	garr_betriebsmeldungen[st_config.i16_meld_startindex + 0] := bm_fuellstand_oeler;
	garr_betriebsmeldungen[st_config.i16_meld_startindex + 1] := FALSE;
	garr_betriebsmeldungen[st_config.i16_meld_startindex + 2] := FALSE;
	garr_betriebsmeldungen[st_config.i16_meld_startindex + 3] := FALSE;
	garr_betriebsmeldungen[st_config.i16_meld_startindex + 4] := FALSE;
	garr_betriebsmeldungen[st_config.i16_meld_startindex + 5] := FALSE;
	garr_betriebsmeldungen[st_config.i16_meld_startindex + 6] := FALSE;
	garr_betriebsmeldungen[st_config.i16_meld_startindex + 7] := FALSE;
	garr_betriebsmeldungen[st_config.i16_meld_startindex + 8] := FALSE;
	garr_betriebsmeldungen[st_config.i16_meld_startindex + 9] := FALSE;
	garr_betriebsmeldungen[st_config.i16_meld_startindex + 10] := FALSE;
	garr_betriebsmeldungen[st_config.i16_meld_startindex + 11] := FALSE;
	garr_betriebsmeldungen[st_config.i16_meld_startindex + 12] := FALSE;
	garr_betriebsmeldungen[st_config.i16_meld_startindex + 13] := FALSE;
	garr_betriebsmeldungen[st_config.i16_meld_startindex + 14] := FALSE;
	garr_betriebsmeldungen[st_config.i16_meld_startindex + 15] := FALSE;
	garr_betriebsmeldungen[st_config.i16_meld_startindex + 16] := FALSE;
	garr_betriebsmeldungen[st_config.i16_meld_startindex + 17] := FALSE;
	garr_betriebsmeldungen[st_config.i16_meld_startindex + 18] := FALSE;
	garr_betriebsmeldungen[st_config.i16_meld_startindex + 19] := FALSE;
END_IF
END_PROGRAM

(* POU Gemeinsamkeiten17xx/Programmbausteine/ST_Schreibe_Persistente_Daten, ST *)
PROGRAM ST_Schreibe_Persistente_Daten
VAR_INPUT
	bExecute			: BOOL;
	bQuit				: BOOL;
	t_schreibintervall		: TIME;
	b_steuerung_ein		: BOOL;
END_VAR
VAR_OUTPUT
	bBusy				: BOOL;
	bError				: BOOL;
	nErrId				: UDINT;
END_VAR
VAR
	fb_write_persistent_data		: FB_WritePersistentData;
	fb_ton_quitt					: TON;
	fb_state_entry				: ST_StateEntry;
	fb_ton_schreiben			: TON;
	fb_get_local_ams_netid		: ST_GetLocalAMSNetID;
	fb_r_trig_execute			: R_TRIG;
	fb_f_trig_steuerung			: F_TRIG;
	sm_fehler_daten_schreiben	: BOOL := FALSE;
	sm_fehler_netid				: BOOL := FALSE;

	gst_manuelles_bestueckprogramm_copy	: struct_bestueckprogramm;
	gst_PersDaten_Copy					: struct_PD;
END_VAR
(* Die Persistenten Daten der Maschine werden in einem wiederkehrenden Zeitintervall in eine Datei im TwinCAT Boot-Ordner geschrieben *)
fb_ton_quitt(IN:= , PT:= t#30s, Q=> , ET=> );
fb_ton_schreiben(IN:= , PT:= t_schreibintervall, Q=> , ET=> );

fb_r_trig_execute(CLK:= bExecute, Q=> );
fb_f_trig_steuerung(CLK:= b_steuerung_ein, Q=> );


fb_state_entry(	i16_pos:= 1 );

CASE fb_state_entry.i16_step OF
(*=======================================================*)
	INIT_OBJ:
		fb_state_entry.i16_next_step := INIT;

(*=======================================================*)
	INIT:
		IF fb_state_entry.E THEN
			bBusy := FALSE;
			bError := FALSE;
			fb_write_persistent_data.START := FALSE;
			fb_ton_schreiben.IN := FALSE;
			fb_get_local_ams_netid.bExecute := FALSE;
			fb_get_local_ams_netid .bQuit := FALSE;
			sm_fehler_daten_schreiben := FALSE;
			sm_fehler_netid := FALSE;
		END_IF

		fb_state_entry.i16_next_step := 20;

(*=======================================================*)
	20:	(* Die AMS-NetID des lokalen PC ermitteln *)
		IF fb_state_entry.E THEN
			fb_get_local_ams_netid.bExecute := TRUE;
		END_IF

		IF fb_get_local_ams_netid.bBusy THEN
			fb_get_local_ams_netid.bExecute := FALSE;
			fb_state_entry.i16_next_step := 30;
		END_IF

(*=======================================================*)
	30:
		IF NOT fb_get_local_ams_netid.bBusy  THEN
			IF NOT fb_get_local_ams_netid.bError THEN
				fb_state_entry.i16_next_step := BEREIT;
			ELSE	(* Fehler *)
				sm_fehler_netid := TRUE;
				fb_state_entry.i16_next_step := FEHLER;
			END_IF
		END_IF

(*=======================================================*)
	BEREIT:	(* Warte auf Freigabeflanke für zyklisches Schreiben der Daten /  Daten sichern, wenn Maschine ausgeschaltet wird *)
		IF 	fb_r_trig_execute.Q OR fb_f_trig_steuerung.Q THEN
			fb_state_entry.i16_next_step := 110;
		END_IF

		(*Schreibe bei einer Änderung*)
		IF	gi16_maschinenstatusinfo <> STATUS_MASCHINE_ARBEITET AND (
			(MEMCMP(ADR(gst_manuelles_bestueckprogramm_copy), ADR(gst_manuelles_bestueckprogramm), SIZEOF(gst_manuelles_bestueckprogramm_copy)) <> 0 ) OR
			(MEMCMP(ADR(gst_PersDaten_Copy), ADR(gst_PersDaten), SIZEOF(gst_PersDaten_Copy)) <> 0 ) 	) THEN
			gst_PersDaten_Copy:=gst_PersDaten;
			gst_manuelles_bestueckprogramm_copy:=gst_manuelles_bestueckprogramm;
			fb_state_entry.i16_next_step := 110;
		END_IF

(*=======================================================*)
	110:	(* Schreibe Persistente Daten *)
		IF fb_state_entry.E THEN
			bBusy := TRUE;
			fb_write_persistent_data.START := TRUE;
		END_IF

		IF fb_write_persistent_data.BUSY THEN
			fb_write_persistent_data.START := FALSE;
			fb_state_entry.i16_next_step := 120;
		END_IF

(*=======================================================*)
	120:	(* Daten wurden geschrieben *)
		IF NOT fb_write_persistent_data.BUSY  THEN
			IF NOT fb_write_persistent_data.ERR THEN
				bBusy := FALSE;
				fb_state_entry.i16_next_step := 100;
			ELSE
				sm_fehler_daten_schreiben := TRUE;
				fb_state_entry.i16_next_step := FEHLER;
			END_IF
		END_IF

(*=======================================================*)
	FEHLER:
		IF fb_state_entry.E THEN
			fb_ton_quitt.IN := TRUE;
			fb_get_local_ams_netid.bExecute := FALSE;
			fb_get_local_ams_netid.bQuit := FALSE;
			bError := TRUE;
		END_IF

		IF  fb_ton_quitt.Q THEN
			fb_ton_quitt.IN := FALSE;
			fb_get_local_ams_netid .bQuit := TRUE;
			fb_state_entry.i16_next_step := INIT;
		END_IF

END_CASE

fb_state_entry(i16_pos:= 2 );

fb_get_local_ams_netid(
	bExecute:= ,
	bQuit:= , 
	bBusy=> , 
	bReady=> , 
	bError=> , 
	nErrId=> , 
	s_ams_netid=> );

fb_write_persistent_data(
	NETID:= '',
	PORT:= 801,
	START:= , 
	TMOUT:= DEFAULT_ADS_TIMEOUT,
	MODE:= SPDM_2PASS,
	BUSY=> , 
	ERR=> , 
	ERRID=> );
END_PROGRAM

(* POU Gemeinsamkeiten17xx/TagReader/ST_Lesen_Schreiben_Tag, ST *)
PROGRAM ST_Lesen_Schreiben_Tag
VAR_INPUT
	st_config					: struct_config;
	st_ctrl_in					: struct_ctrl_in;
END_VAR
VAR_OUTPUT
	st_ctrl_out				: struct_ctrl_out;
END_VAR
VAR
	fb_r_trig_lesen			: R_TRIG;
	fb_r_trig_schreiben		: R_TRIG;
	fb_r_trig_WT_ruecksetzen	: R_TRIG;
	fb_r_trig_auto_lesen		: R_TRIG;
	fb_ton_lesen				: TON;
	fb_ton_auto_lesen				: TON;
	fb_ton_Timeout				: TON;

	fb_state_entry				: ST_StateEntry;
	fb_ton_quitt				: TON;
	fb_r_trig_quittieren			: R_TRIG;
	fb_ton_uez				: TON;

	sm_WT_Nummer_ungueltig				: BOOL := FALSE;
	sm_wt_hat_kein_tag					: BOOL := FALSE;
	bm_kein_WT_im_Aktionsfeld			: BOOL := FALSE;
	bm_Wert_nicht_erlaubt					: BOOL := FALSE;

	i									: INT;

	i16_betriebsart: BOOL;
END_VAR
fb_ton_quitt(IN:= , PT:= t#500ms, Q=> , ET=> );
fb_ton_uez(IN:= , PT:= , Q=>  , ET=> );

fb_ton_lesen(IN:= , PT:= t#500ms, Q=> , ET=> );
fb_r_trig_lesen(CLK:=visu.st_tagreader.b_start_lesen , Q=>);
fb_ton_auto_lesen(IN:=balluff_tag_reader.fb.e_tag_im_aktionsfeld   AND gi16_betriebsart = HAND , PT:= t#500ms, Q=> , ET=> );
fb_r_trig_auto_lesen(CLK:= fb_ton_auto_lesen.Q , Q=>);


fb_r_trig_schreiben(CLK:=visu.st_tagreader.b_start_schreiben , Q=>);
fb_r_trig_WT_ruecksetzen(CLK:=visu.st_tagreader.b_WT_ruecksetzen , Q=>);

visu.st_tagreader.b_tag_im_Aktionsfeld:=balluff_tag_reader.fb.e_tag_im_aktionsfeld;

fb_state_entry(
	i16_next_step:= ,
	i16_pos:= 1,
	s_debugtext:= ,
	E=> ,
	X=> ,
	i16_step=> ,
	i16_last_step=> );

(*wenn Tagreader nicht bereit ist stoppen*)
IF	Balluff_Tag_Reader.fb.fb_state_entry.i16_step<BEREIT OR
	Balluff_Tag_Reader.fb.fb_state_entry.i16_step>=STOP THEN
	fb_state_entry.i16_next_step := STOP;
END_IF

fb_ton_Timeout(IN:= fb_state_entry.i16_step>BEREIT AND fb_state_entry.i16_step<FEHLER, PT:= t#35s, Q=> , ET=> );
IF	fb_ton_Timeout.Q THEN
	fb_state_entry.i16_next_step := FEHLER;
END_IF

CASE fb_state_entry.i16_step OF
(*=======================================================*)
	INIT_OBJ:

		fb_state_entry.i16_next_step := INIT;

(*=======================================================*)
	INIT:
		IF 	fb_state_entry.E THEN
			balluff_tag_reader.st_ctrl.in.b_start_lesen := FALSE;
			balluff_tag_reader.st_ctrl.in.b_start_schreiben := FALSE;

			sm_WT_Nummer_ungueltig:=FALSE;
			sm_wt_hat_kein_tag:=FALSE;

			visu.st_tagreader.b_WT_ruecksetzen:=FALSE;
			visu.st_tagreader.b_start_schreiben:=FALSE;
			visu.st_tagreader.b_start_lesen:=FALSE;
		END_IF

		(*-----------------------Weiterschaltbedingungen----------------------------*)
		fb_state_entry.i16_next_step := BEREIT;

(*=======================================================*)
	BEREIT:	(* Warte auf Start von Kontroller *)

		(*-----------------------Weiterschaltbedingungen----------------------------*)
		IF	balluff_tag_reader.fb.e_tag_im_aktionsfeld   AND gi16_betriebsart = HAND THEN
			IF	fb_r_trig_lesen.Q  OR fb_r_trig_auto_lesen.Q THEN
				fb_state_entry.i16_next_step := 120;
			END_IF

			IF	fb_r_trig_schreiben.Q THEN
				fb_state_entry.i16_next_step := 150;
			END_IF

			IF	fb_r_trig_WT_ruecksetzen.Q THEN
				fb_state_entry.i16_next_step := 200;
			END_IF
		ELSE
			IF	fb_r_trig_WT_ruecksetzen.Q OR
				fb_r_trig_schreiben.Q OR
				fb_r_trig_lesen.Q THEN
				fb_state_entry.i16_next_step := 110;
			END_IF
		END_IF

(*=======================================================*)
	110:
		IF 	fb_state_entry.E THEN
			fb_ton_uez.PT:=t#2000ms ;
			fb_ton_uez.IN:=TRUE ;
			bm_kein_WT_im_Aktionsfeld:=TRUE;
		END_IF

		(*-----------------------Weiterschaltbedingungen----------------------------*)
		IF	fb_ton_uez.Q THEN
			fb_state_entry.i16_next_step := INIT;
			fb_ton_uez.IN:=FALSE ;
			bm_kein_WT_im_Aktionsfeld:=FALSE;
		END_IF

(*=======================================================*)
	120:
		IF 	fb_state_entry.E THEN
			gst_tag_data.Articelnumber:='LESEN';
			gst_tag_data.LastUsedTool:=0;
			IF gst_datensatz.st_md.i16_tag_data_structur_version = 0 THEN
				gst_tag_data.StateParts[0]:=100;
				gst_tag_data.StateParts[1]:=100;
			ELSIF gst_datensatz.st_md.i16_tag_data_structur_version = 1 THEN
				FOR i:= 0 TO 7 BY 1 DO
					gst_tag_data.StateParts[i] := 100;
				END_FOR
			END_IF
			gst_tag_data.WpcNumber:=0;
			fb_ton_lesen.IN:=TRUE;
		END_IF

	(*-----------------------Weiterschaltbedingungen----------------------------*)
	IF	fb_ton_lesen.Q THEN
		fb_ton_lesen.IN:=FALSE;
		fb_state_entry.i16_next_step := 130;
	END_IF

(*=======================================================*)
	130: (* WT-Tag mit RFID-Lesegerät auslesen *)
		IF 	fb_state_entry.E THEN
			balluff_tag_reader.st_ctrl.in.b_start_lesen := TRUE;
			balluff_tag_reader.fb.i16_addresse := 0;
			balluff_tag_reader.fb.i16_anzahl_byte := SIZEOF(gst_tag_data);
		END_IF

		(*-----------------------Weiterschaltbedingungen----------------------------*)
		IF 	balluff_tag_reader.st_ctrl.out.b_fertig AND NOT fb_state_entry.E THEN
			IF gst_datensatz.st_md.i16_tag_data_structur_version = 0 THEN
				gst_tag_data.WpcNumber := balluff_tag_reader.fb.s_lese_daten[0];
				gst_tag_data.StateParts[0] := balluff_tag_reader.fb.s_lese_daten[1];
				gst_tag_data.StateParts[1] := balluff_tag_reader.fb.s_lese_daten[2];

				MEMCPY( ADR(gst_tag_data.Articelnumber), ADR(balluff_tag_reader.fb.s_lese_daten[3]), 50);
				gst_tag_data.LastUsedTool := balluff_tag_reader.fb.s_lese_daten[54];
				MEMCPY( ADR(gst_tag_data.UmlNo_VPE), ADR(balluff_tag_reader.fb.s_lese_daten[55]), 4);

				(*gst_datensatz.st_md.s_aktuelle_artikelnummer := gst_tag_data.Articelnumber;*)
			ELSIF gst_datensatz.st_md.i16_tag_data_structur_version = 1 THEN
				gst_tag_data.WpcNumber := balluff_tag_reader.fb.s_lese_daten[0];
				FOR i:= 0 TO 7 BY 1 DO
					gst_tag_data.StateParts[i] := balluff_tag_reader.fb.s_lese_daten[i + 1];
				END_FOR
				gst_tag_data.AmountPartsOnWpc := balluff_tag_reader.fb.s_lese_daten[10];
				gst_tag_data.LastUsedTool := balluff_tag_reader.fb.s_lese_daten[15];
				MEMCPY( ADR(gst_tag_data.Articelnumber), ADR(balluff_tag_reader.fb.s_lese_daten[20]), 50);
				MEMCPY( ADR(gst_tag_data.UmlNo_VPE), ADR(balluff_tag_reader.fb.s_lese_daten[71]), 4);
			END_IF

			IF 	gst_tag_data.WpcNumber >= 0 AND gst_tag_data.WpcNumber <=50 THEN
				balluff_tag_reader.st_ctrl.in.b_start_lesen := FALSE;
				fb_state_entry.i16_next_step := INIT;
			ELSE
				(* Fehler: Tagnummer ist nicht im gültigem Bereich *)
				balluff_tag_reader.st_ctrl.in.b_start_lesen := FALSE;
				sm_WT_Nummer_ungueltig := TRUE;
				fb_state_entry.i16_next_step := FEHLER;
			END_IF
		END_IF

(*=======================================================*)
	150:	(*Artikelnummer schreiben*)
		IF 	fb_state_entry.E THEN
			IF gst_datensatz.st_md.i16_tag_data_structur_version = 0 THEN
				balluff_tag_reader.st_ctrl.in.b_start_schreiben := TRUE;
	
				balluff_tag_reader.fb.i16_addresse := 3;
				balluff_tag_reader.fb.i16_anzahl_byte := SIZEOF(gst_tag_data.Articelnumber);
				MEMCPY(ADR(balluff_tag_reader.fb.s_schreib_daten),ADR(gst_tag_data.Articelnumber),  50);
			ELSIF gst_datensatz.st_md.i16_tag_data_structur_version = 1 THEN
				balluff_tag_reader.st_ctrl.in.b_start_schreiben := TRUE;
	
				balluff_tag_reader.fb.i16_addresse := 20;
				balluff_tag_reader.fb.i16_anzahl_byte := SIZEOF(gst_tag_data.Articelnumber);
				MEMCPY(ADR(balluff_tag_reader.fb.s_schreib_daten),ADR(gst_tag_data.Articelnumber),  50);
			END_IF
		END_IF

		(*-----------------------Weiterschaltbedingungen----------------------------*)
		IF 	balluff_tag_reader.st_ctrl.out.b_fertig AND NOT fb_state_entry.E THEN
			(* Ok: Daten sind auf dem Tag *)
			balluff_tag_reader.st_ctrl.in.b_start_schreiben := FALSE;
			fb_state_entry.i16_next_step := 155;
		END_IF

(*=======================================================*)
	155:	(*UML_Stueckzaehler schreiben*)
		IF 	fb_state_entry.E THEN
			IF gst_datensatz.st_md.i16_tag_data_structur_version = 0 THEN
				balluff_tag_reader.st_ctrl.in.b_start_schreiben := TRUE;

				balluff_tag_reader.fb.i16_addresse := 55;
				balluff_tag_reader.fb.i16_anzahl_byte := SIZEOF(gst_tag_data.UmlNo_VPE);
				MEMCPY( ADR(balluff_tag_reader.fb.s_schreib_daten), ADR(gst_tag_data.UmlNo_VPE), 4);

			ELSIF gst_datensatz.st_md.i16_tag_data_structur_version = 1 THEN
				balluff_tag_reader.st_ctrl.in.b_start_schreiben := TRUE;

				balluff_tag_reader.fb.i16_addresse := 71;
				balluff_tag_reader.fb.i16_anzahl_byte := SIZEOF(gst_tag_data.UmlNo_VPE);
				MEMCPY(ADR(balluff_tag_reader.fb.s_schreib_daten),ADR(gst_tag_data.UmlNo_VPE),  4);
			END_IF
		END_IF

		(*-----------------------Weiterschaltbedingungen----------------------------*)
		IF 	balluff_tag_reader.st_ctrl.out.b_fertig AND NOT fb_state_entry.E THEN
			(* Ok: Daten sind auf dem Tag *)
			balluff_tag_reader.st_ctrl.in.b_start_schreiben := FALSE;
			fb_state_entry.i16_next_step := 160;
		END_IF

(*=======================================================*)
	160:	(*States schreiben*)
		IF 	fb_state_entry.E THEN
			IF gst_datensatz.st_md.i16_tag_data_structur_version = 0 THEN
				balluff_tag_reader.st_ctrl.in.b_start_schreiben := TRUE;
	
				balluff_tag_reader.fb.i16_addresse := 1;
				balluff_tag_reader.fb.i16_anzahl_byte := 2;
				balluff_tag_reader.fb.s_schreib_daten[0] := DINT_TO_BYTE(gst_tag_data.StateParts[0]);
				balluff_tag_reader.fb.s_schreib_daten[1] := DINT_TO_BYTE(gst_tag_data.StateParts[1]);
			ELSIF gst_datensatz.st_md.i16_tag_data_structur_version = 1 THEN
				balluff_tag_reader.st_ctrl.in.b_start_schreiben := TRUE;
	
				balluff_tag_reader.fb.i16_addresse := 1;
				balluff_tag_reader.fb.i16_anzahl_byte := 8;
				FOR i:= 0 TO 7 BY 1 DO
					balluff_tag_reader.fb.s_schreib_daten[i] := DINT_TO_BYTE(gst_tag_data.StateParts[i]);
				END_FOR
			END_IF
		END_IF

		(*-----------------------Weiterschaltbedingungen----------------------------*)
		IF balluff_tag_reader.st_ctrl.out.b_fertig AND NOT fb_state_entry.E THEN
			(* Ok: Daten sind auf dem Tag *)
			balluff_tag_reader.st_ctrl.in.b_start_schreiben := FALSE;
			fb_state_entry.i16_next_step := 170;
		END_IF

(*=======================================================*)
	170:	(* WT Nummer schreiben *)
		IF	 fb_state_entry.E THEN
			(* Starte Schreib Prozess *)
			balluff_tag_reader.fb.i16_addresse := 0;
			balluff_tag_reader.fb.i16_anzahl_byte := 1;
			balluff_tag_reader.fb.s_schreib_daten[0] := gst_tag_data.WpcNumber;
			balluff_tag_reader.st_ctrl.in.b_start_schreiben := TRUE;
		END_IF

		(*-----------------------Weiterschaltbedingungen----------------------------*)
		IF 	balluff_tag_reader.st_ctrl.out.b_fertig AND NOT fb_state_entry.E THEN
			balluff_tag_reader.st_ctrl.in.b_start_schreiben := FALSE;
			fb_state_entry.i16_next_step := 180;
		END_IF

(*=======================================================*)
	180:	(* letztes benutzes Werkzeug schreiben*)
		IF 	fb_state_entry.E THEN
			(* Starte Schreib Prozess *)
			IF gst_datensatz.st_md.i16_tag_data_structur_version = 0 THEN
				balluff_tag_reader.fb.i16_addresse := 54;
				balluff_tag_reader.fb.i16_anzahl_byte := 1;
				balluff_tag_reader.fb.s_schreib_daten[0] := gst_tag_data.LastUsedTool;
				balluff_tag_reader.st_ctrl.in.b_start_schreiben := TRUE;
			ELSIF gst_datensatz.st_md.i16_tag_data_structur_version = 1 THEN
				balluff_tag_reader.fb.i16_addresse := 15;
				balluff_tag_reader.fb.i16_anzahl_byte := 1;
				balluff_tag_reader.fb.s_schreib_daten[0] := gst_tag_data.LastUsedTool;
				balluff_tag_reader.st_ctrl.in.b_start_schreiben := TRUE;
			END_IF
		END_IF

		(*-----------------------Weiterschaltbedingungen----------------------------*)
		IF 	balluff_tag_reader.st_ctrl.out.b_fertig AND NOT fb_state_entry.E THEN
			balluff_tag_reader.st_ctrl.in.b_start_schreiben := FALSE;
			IF gst_datensatz.st_md.i16_tag_data_structur_version = 0 THEN
				fb_state_entry.i16_next_step := 120;
			ELSIF gst_datensatz.st_md.i16_tag_data_structur_version = 1 THEN
				fb_state_entry.i16_next_step := 190;
			END_IF
		END_IF

(*=======================================================*)
	190:	(* Anzahl ISK auf WT *)
		IF 	fb_state_entry.E THEN
			(* Starte Schreib Prozess *)
			balluff_tag_reader.fb.i16_addresse := 10;
			balluff_tag_reader.fb.i16_anzahl_byte := 1;
			balluff_tag_reader.fb.s_schreib_daten[0] := gst_tag_data.AmountPartsOnWpc;
			balluff_tag_reader.st_ctrl.in.b_start_schreiben := TRUE;
		END_IF

		(*-----------------------Weiterschaltbedingungen----------------------------*)
		IF 	balluff_tag_reader.st_ctrl.out.b_fertig AND NOT fb_state_entry.E THEN
			balluff_tag_reader.st_ctrl.in.b_start_schreiben := FALSE;
			fb_state_entry.i16_next_step := 120;
		END_IF

(*=======================================================*)
	200:	(*WT zurücksetzen*)
		IF	 fb_state_entry.E THEN
			IF gst_datensatz.st_md.i16_tag_data_structur_version = 0 THEN
				gst_tag_data.StateParts[0] := PART_NO;
				gst_tag_data.StateParts[1] := PART_NO;

				balluff_tag_reader.st_ctrl.in.b_start_schreiben := TRUE;
				balluff_tag_reader.fb.i16_addresse := 1;
				balluff_tag_reader.fb.i16_anzahl_byte := 2;
				balluff_tag_reader.fb.s_schreib_daten[0] := DINT_TO_BYTE(gst_tag_data.StateParts[0]);
				balluff_tag_reader.fb.s_schreib_daten[1] := DINT_TO_BYTE(gst_tag_data.StateParts[1]);
			ELSIF gst_datensatz.st_md.i16_tag_data_structur_version = 1 THEN
				FOR i:= 0 TO 7 BY 1 DO
					gst_tag_data.StateParts[i] := PART_NO;
				END_FOR
	
				balluff_tag_reader.st_ctrl.in.b_start_schreiben := TRUE;
				balluff_tag_reader.fb.i16_addresse := 1;
				balluff_tag_reader.fb.i16_anzahl_byte := 8;
				FOR i:= 0 TO 7 BY 1 DO
					balluff_tag_reader.fb.s_schreib_daten[i] := DINT_TO_BYTE(gst_tag_data.StateParts[i]);
				END_FOR
			END_IF
		END_IF

		(*-----------------------Weiterschaltbedingungen----------------------------*)
		IF 	balluff_tag_reader.st_ctrl.out.b_fertig AND NOT fb_state_entry.E THEN
			(* Ok: Daten sind auf dem Tag *)
			balluff_tag_reader.st_ctrl.in.b_start_schreiben := FALSE;
			fb_state_entry.i16_next_step := 210;
		END_IF

(*=======================================================*)
	210:	(* letztes benutzes Werkzeug schreiben*)
		IF 	fb_state_entry.E THEN
			gst_tag_data.LastUsedTool := 0;
			(* Starte Schreib Prozess *)
			IF gst_datensatz.st_md.i16_tag_data_structur_version = 0 THEN
				balluff_tag_reader.fb.i16_addresse := 54;
				balluff_tag_reader.fb.i16_anzahl_byte := 1;
				balluff_tag_reader.fb.s_schreib_daten[0] := 0;
				balluff_tag_reader.st_ctrl.in.b_start_schreiben := TRUE;
			ELSIF gst_datensatz.st_md.i16_tag_data_structur_version = 1 THEN
				balluff_tag_reader.fb.i16_addresse := 15;
				balluff_tag_reader.fb.i16_anzahl_byte := 1;
				balluff_tag_reader.fb.s_schreib_daten[0] := 0;
				balluff_tag_reader.st_ctrl.in.b_start_schreiben := TRUE;
			END_IF
		END_IF

		(*-----------------------Weiterschaltbedingungen----------------------------*)
		IF 	balluff_tag_reader.st_ctrl.out.b_fertig AND NOT fb_state_entry.E THEN
			balluff_tag_reader.st_ctrl.in.b_start_schreiben := FALSE;
			fb_state_entry.i16_next_step := INIT;
		END_IF

(*=======================================================*)
	FEHLER:
		IF 	fb_state_entry.E THEN
			st_ctrl_out.b_fehler := TRUE;
			fb_ton_quitt.IN := FALSE;
		END_IF

		(*-----------------------Weiterschaltbedingungen----------------------------*)
		IF 	st_ctrl_in.b_quitt AND NOT fb_state_entry.E THEN
			st_ctrl_out.b_fehler := FALSE;
			fb_ton_quitt.IN := TRUE;
		END_IF

		IF 	fb_ton_quitt.Q THEN
			fb_ton_quitt.IN := FALSE;
			fb_state_entry.i16_next_step := INIT;
		END_IF

(*=======================================================*)
	STOP:
		IF 	fb_state_entry.E THEN
			;
		END_IF

		(*-----------------------Weiterschaltbedingungen----------------------------*)
		IF 	Balluff_Tag_Reader.fb.fb_state_entry.i16_step=BEREIT THEN
			fb_state_entry.i16_next_step := INIT;
		END_IF

END_CASE

fb_state_entry(
	i16_next_step:= ,
	i16_pos:= 2,
	s_debugtext:= ,
	E=> ,
	X=> ,
	i16_step=> ,
	i16_last_step=> );

(* Fehlermeldungen ab dem Startindex in das globale Störmeldungsarray schreiben *)
garr_stoermeldungen[st_config.i16_meld_startindex + 0] := sm_WT_Nummer_ungueltig;
garr_stoermeldungen[st_config.i16_meld_startindex + 1] := sm_wt_hat_kein_tag;
garr_stoermeldungen[st_config.i16_meld_startindex + 2] :=FALSE;
garr_stoermeldungen[st_config.i16_meld_startindex + 3] := FALSE;
garr_stoermeldungen[st_config.i16_meld_startindex + 4] := FALSE;
garr_stoermeldungen[st_config.i16_meld_startindex + 5] := FALSE;
garr_stoermeldungen[st_config.i16_meld_startindex + 6] := FALSE;
garr_stoermeldungen[st_config.i16_meld_startindex + 7] := FALSE;
garr_stoermeldungen[st_config.i16_meld_startindex + 8] := FALSE;
garr_stoermeldungen[st_config.i16_meld_startindex + 9] := FALSE;
garr_stoermeldungen[st_config.i16_meld_startindex + 10] := FALSE;
garr_stoermeldungen[st_config.i16_meld_startindex + 11] := FALSE;
garr_stoermeldungen[st_config.i16_meld_startindex + 12] := FALSE;
garr_stoermeldungen[st_config.i16_meld_startindex + 13] := FALSE;
garr_stoermeldungen[st_config.i16_meld_startindex + 14] := FALSE;
garr_stoermeldungen[st_config.i16_meld_startindex + 15] := FALSE;
garr_stoermeldungen[st_config.i16_meld_startindex + 16] := FALSE;
garr_stoermeldungen[st_config.i16_meld_startindex + 17] := FALSE;
garr_stoermeldungen[st_config.i16_meld_startindex + 18] := FALSE;
garr_stoermeldungen[st_config.i16_meld_startindex + 19] := FALSE;

garr_betriebsmeldungen[st_config.i16_meld_startindex + 0] := bm_kein_WT_im_Aktionsfeld;
garr_betriebsmeldungen[st_config.i16_meld_startindex + 1] := bm_Wert_nicht_erlaubt;
garr_betriebsmeldungen[st_config.i16_meld_startindex + 2] := FALSE;
garr_betriebsmeldungen[st_config.i16_meld_startindex + 3] := FALSE;
garr_betriebsmeldungen[st_config.i16_meld_startindex + 4] := FALSE;
garr_betriebsmeldungen[st_config.i16_meld_startindex + 5] := FALSE;
garr_betriebsmeldungen[st_config.i16_meld_startindex + 6] := FALSE;
garr_betriebsmeldungen[st_config.i16_meld_startindex + 7] := FALSE;
garr_betriebsmeldungen[st_config.i16_meld_startindex + 8] := FALSE;
garr_betriebsmeldungen[st_config.i16_meld_startindex + 9] := FALSE;
garr_betriebsmeldungen[st_config.i16_meld_startindex + 10] := FALSE;
garr_betriebsmeldungen[st_config.i16_meld_startindex + 11] := FALSE;
garr_betriebsmeldungen[st_config.i16_meld_startindex + 12] := FALSE;
garr_betriebsmeldungen[st_config.i16_meld_startindex + 13] := FALSE;
garr_betriebsmeldungen[st_config.i16_meld_startindex + 14] := FALSE;
garr_betriebsmeldungen[st_config.i16_meld_startindex + 15] := FALSE;
garr_betriebsmeldungen[st_config.i16_meld_startindex + 16] := FALSE;
garr_betriebsmeldungen[st_config.i16_meld_startindex + 17] := FALSE;
garr_betriebsmeldungen[st_config.i16_meld_startindex + 18] := FALSE;
garr_betriebsmeldungen[st_config.i16_meld_startindex + 19] := FALSE;
END_PROGRAM

(* POU Gemeinsamkeiten17xx/Visu/ST_VisuRouter, ST *)
PROGRAM ST_VisuRouter
VAR
END_VAR
(*Anzeige der aktuellen Betriebsart*)
CASE gi16_betriebsart OF
	KEINE:
		visu_hinten.in.betriebsart := visu_hinten.in.texte.txt_variabel[8];

	AUTO:
		visu_hinten.in.betriebsart := visu_hinten.in.texte.txt_variabel[5];

	TIPPEN:
		visu_hinten.in.betriebsart := visu_hinten.in.texte.txt_variabel[6];

	HAND:
		visu_hinten.in.betriebsart := visu_hinten.in.texte.txt_variabel[7];
END_CASE

(*Anzeige des Maschinenstatus*)
CASE gi16_maschinenstatusinfo OF
	KEIN_STATUS:
		visu_hinten.in.s_maschinenstatusinfo := visu_hinten.in.texte.txt_variabel[0];

	STATUS_FEHLER:
		visu_hinten.in.s_maschinenstatusinfo := visu_hinten.in.texte.txt_variabel[1];

	STATUS_FEHLER_QUITTIERT:
		visu_hinten.in.s_maschinenstatusinfo := visu_hinten.in.texte.txt_variabel[2];

	STATUS_BETRIEBSBEREIT:
		visu_hinten.in.s_maschinenstatusinfo := visu_hinten.in.texte.txt_variabel[3];

	STATUS_MASCHINE_ARBEITET:
		visu_hinten.in.s_maschinenstatusinfo := visu_hinten.in.texte.txt_variabel[4];
END_CASE

visu_hinten.in.i16_maschinenstatusinfo := gi16_maschinenstatusinfo;
visu_hinten.in.s_betriebsmeldung := ST_Virtuelle_Masterachse.bm_an_visu_hinten;
visu_hinten.in.i16_position_ist := LREAL_TO_INT(bestueckachse.NcToPlc.ModuloActPos);
visu_hinten.in.i16_typ_zelle := gst_datensatz.st_md.i16_typ_zelle;
visu_hinten.in.i16_typ_bandeinzug:=gst_datensatz.st_wkz.i16_typ_bandeinzug;
visu_hinten.in.band_ID_Puffer_aus:=gst_datensatz.st_md.b_band_ID_Puffer_aus;


visu_hinten.in.texte.txt_zylindernamen[2].s_einfahren:=visu_hinten.in.texte.txt_zylindernamen[0].s_einfahren;
visu_hinten.in.texte.txt_zylindernamen[2].s_ausfahren:=visu_hinten.in.texte.txt_zylindernamen[0].s_ausfahren;
visu_hinten.in.texte.txt_zylindernamen[3].s_einfahren:=visu_hinten.in.texte.txt_zylindernamen[1].s_einfahren;
visu_hinten.in.texte.txt_zylindernamen[3].s_ausfahren:=visu_hinten.in.texte.txt_zylindernamen[1].s_ausfahren;

CASE gst_datensatz.st_md.i16_typ_zelle OF
	KEINE_ZELLE:
		;

	BESTUECKZELLE_1700:

		CASE gst_datensatz.st_wkz.i16_typ_bandeinzug OF
			KEIN_EINZUG:
				;

			STANDARD_2FACH_V2:
				;

			 SERVO:
				(* Die Seitenbezeichnungen (links, rechts) beziehen sich auf die Maschinenvorderseite *)
				(* Haspel Links Heben *)
				zyl_haspel_li_heben.fb.b_direkttaste_ausfahren := visu_hinten.out.zylinder_direkttasten[0].b_ausfahren;
				zyl_haspel_li_heben.fb.b_direkttaste_einfahren := visu_hinten.out.zylinder_direkttasten[0].b_einfahren;
				visu_hinten.in.zylinder_sensoren[0].b_eingefahren := zyl_haspel_li_heben.fb.e_sensor1_eingefahren;
				visu_hinten.in.zylinder_sensoren[0].b_ausgefahren := zyl_haspel_li_heben.fb.e_sensor1_ausgefahren;

				(* Haspel Links Sperren *)
				zyl_haspel_li_sperren.fb.b_direkttaste_ausfahren := visu_hinten.out.zylinder_direkttasten[1].b_ausfahren;
				zyl_haspel_li_sperren.fb.b_direkttaste_einfahren :=  visu_hinten.out.zylinder_direkttasten[1].b_einfahren;
				zyl_haspel_li_abspulen.fb.b_direkttaste_ausfahren:=visu_hinten.out.zylinder_direkttasten[1].b_einfahren; (*Abspulzylinder beim Entriegeln anheben*)
				visu_hinten.in.zylinder_sensoren[1].b_eingefahren := zyl_haspel_li_sperren.fb.e_sensor1_eingefahren;
				visu_hinten.in.zylinder_sensoren[1].b_ausgefahren := zyl_haspel_li_sperren.fb.e_sensor1_ausgefahren;
		
				(* Haspel Rechts Heben *)
				zyl_haspel_re_heben.fb.b_direkttaste_ausfahren := visu_hinten.out.zylinder_direkttasten[2].b_ausfahren;
				zyl_haspel_re_heben.fb.b_direkttaste_einfahren := visu_hinten.out.zylinder_direkttasten[2].b_einfahren;
				visu_hinten.in.zylinder_sensoren[2].b_eingefahren := zyl_haspel_re_heben.fb.e_sensor1_eingefahren;
				visu_hinten.in.zylinder_sensoren[2].b_ausgefahren := zyl_haspel_re_heben.fb.e_sensor1_ausgefahren;
		
				(* Haspel Rechts Sperren *)
				zyl_haspel_re_sperren.fb.b_direkttaste_ausfahren := visu_hinten.out.zylinder_direkttasten[3].b_ausfahren;
				zyl_haspel_re_sperren.fb.b_direkttaste_einfahren := visu_hinten.out.zylinder_direkttasten[3].b_einfahren;
				zyl_haspel_re_abspulen.fb.b_direkttaste_ausfahren:=visu_hinten.out.zylinder_direkttasten[3].b_einfahren; (*Abspulzylinder beim Entriegeln anheben*)
				visu_hinten.in.zylinder_sensoren[3].b_eingefahren := zyl_haspel_re_sperren.fb.e_sensor1_eingefahren;
				visu_hinten.in.zylinder_sensoren[3].b_ausgefahren := zyl_haspel_re_sperren.fb.e_sensor1_ausgefahren;
		
				(* Bandfänger *)
				zyl_bandfaenger.fb.b_direkttaste_ausfahren := visu_hinten.out.zylinder_direkttasten[4].b_ausfahren;
				zyl_bandfaenger.fb.b_direkttaste_einfahren := visu_hinten.out.zylinder_direkttasten[4].b_einfahren;
				visu_hinten.in.zylinder_sensoren[4].b_eingefahren := zyl_bandfaenger.fb.e_sensor1_eingefahren;
				visu_hinten.in.zylinder_sensoren[4].b_ausgefahren := zyl_bandfaenger.fb.e_sensor1_ausgefahren;
		
				(* Bandklemmen *)
				zyl_bandklemmen.fb.b_direkttaste_ausfahren := visu_hinten.out.zylinder_direkttasten[5].b_ausfahren;
				zyl_bandklemmen.fb.b_direkttaste_einfahren := visu_hinten.out.zylinder_direkttasten[5].b_einfahren;
				visu_hinten.in.zylinder_sensoren[5].b_eingefahren := zyl_bandklemmen.fb.e_sensor1_eingefahren;
				visu_hinten.in.zylinder_sensoren[5].b_ausgefahren := zyl_bandklemmen.fb.e_sensor1_ausgefahren;
		
				(* Bandwechselhalter links *)
				zyl_bawe_halter_li.fb.b_direkttaste_ausfahren := visu_hinten.out.zylinder_direkttasten[6].b_ausfahren;
				zyl_bawe_halter_li.fb.b_direkttaste_einfahren := visu_hinten.out.zylinder_direkttasten[6].b_einfahren;
				visu_hinten.in.zylinder_sensoren[6].b_eingefahren := zyl_bawe_halter_li.fb.e_sensor1_eingefahren;
				visu_hinten.in.zylinder_sensoren[6].b_ausgefahren := zyl_bawe_halter_li.fb.e_sensor1_ausgefahren;
		
				(* Bandwechselhalter rechts *)
				zyl_bawe_halter_re.fb.b_direkttaste_ausfahren := visu_hinten.out.zylinder_direkttasten[7].b_ausfahren;
				zyl_bawe_halter_re.fb.b_direkttaste_einfahren := visu_hinten.out.zylinder_direkttasten[7].b_einfahren;
				visu_hinten.in.zylinder_sensoren[7].b_eingefahren := zyl_bawe_halter_re.fb.e_sensor1_eingefahren;
				visu_hinten.in.zylinder_sensoren[7].b_ausgefahren := zyl_bawe_halter_re.fb.e_sensor1_ausgefahren;
		
				(* Bandwechselfänger links *)
				zyl_bawe_faenger_li.fb.b_direkttaste_ausfahren := visu_hinten.out.zylinder_direkttasten[8].b_ausfahren;
				zyl_bawe_faenger_li.fb.b_direkttaste_einfahren := visu_hinten.out.zylinder_direkttasten[8].b_einfahren;
				visu_hinten.in.zylinder_sensoren[8].b_eingefahren := zyl_bawe_faenger_li.fb.e_sensor1_eingefahren;
				visu_hinten.in.zylinder_sensoren[8].b_ausgefahren := zyl_bawe_faenger_li.fb.e_sensor1_ausgefahren;
		
				(* Bandwechselfänger rechts *)
				zyl_bawe_faenger_re.fb.b_direkttaste_ausfahren := visu_hinten.out.zylinder_direkttasten[9].b_ausfahren;
				zyl_bawe_faenger_re.fb.b_direkttaste_einfahren := visu_hinten.out.zylinder_direkttasten[9].b_einfahren;
				visu_hinten.in.zylinder_sensoren[9].b_eingefahren := zyl_bawe_faenger_re.fb.e_sensor1_eingefahren;
				visu_hinten.in.zylinder_sensoren[9].b_ausgefahren := zyl_bawe_faenger_re.fb.e_sensor1_ausgefahren;

				(*Spulenwechsel bie 1700======================*)
				(*Quervorschub*)
				zyl_bawe_querschub.st_ctrl.in.b_ausfahren := visu_hinten.out.zylinder_direkttasten[12].b_ausfahren;
				zyl_bawe_querschub.st_ctrl.in.b_einfahren := visu_hinten.out.zylinder_direkttasten[12].b_einfahren;

				visu_hinten.in.zylinder_sensoren[12].b_eingefahren := zyl_bawe_querschub.fb.e_sensor1_eingefahren;
				visu_hinten.in.zylinder_sensoren[12].b_ausgefahren := zyl_bawe_querschub.fb.e_sensor1_ausgefahren;

				(*Haspel verschieben*)
				zyl_haspel_verschieben.st_ctrl.in.b_ausfahren := visu_hinten.out.zylinder_direkttasten[13].b_ausfahren;
				zyl_haspel_verschieben.st_ctrl.in.b_einfahren := visu_hinten.out.zylinder_direkttasten[13].b_einfahren;

				visu_hinten.in.zylinder_sensoren[13].b_eingefahren := zyl_haspel_verschieben.fb.e_sensor1_eingefahren;
				visu_hinten.in.zylinder_sensoren[13].b_ausgefahren := zyl_haspel_verschieben.fb.e_sensor1_ausgefahren;

				(*Bandeinzug verschieben*)
				zyl_bandeinzuege_verschieben.st_ctrl.in.b_ausfahren := visu_hinten.out.zylinder_direkttasten[14].b_ausfahren;
				zyl_bandeinzuege_verschieben.st_ctrl.in.b_einfahren := visu_hinten.out.zylinder_direkttasten[14].b_einfahren;

				visu_hinten.in.zylinder_sensoren[14].b_eingefahren := zyl_bandeinzuege_verschieben.fb.e_sensor1_eingefahren;
				visu_hinten.in.zylinder_sensoren[14].b_ausgefahren := zyl_bandeinzuege_verschieben.fb.e_sensor1_ausgefahren;

				(* Haspel Links abspulen *)
				zyl_haspel_li_abspulen.fb.b_direkttaste_ausfahren := visu_hinten.out.zylinder_direkttasten[15].b_ausfahren;
				zyl_haspel_li_abspulen.fb.b_direkttaste_einfahren := visu_hinten.out.zylinder_direkttasten[15].b_einfahren;
				visu_hinten.in.zylinder_sensoren[15].b_eingefahren := NOT zyl_haspel_li_abspulen.fb.e_sensor1_ausgefahren;
				visu_hinten.in.zylinder_sensoren[15].b_ausgefahren := zyl_haspel_li_abspulen.fb.e_sensor1_ausgefahren;

				(* Haspel Rechts abspulen *)
				zyl_haspel_re_abspulen.fb.b_direkttaste_ausfahren := visu_hinten.out.zylinder_direkttasten[16].b_ausfahren;
				zyl_haspel_re_abspulen.fb.b_direkttaste_einfahren := visu_hinten.out.zylinder_direkttasten[16].b_einfahren;
				visu_hinten.in.zylinder_sensoren[16].b_eingefahren := NOT zyl_haspel_re_abspulen.fb.e_sensor1_ausgefahren;
				visu_hinten.in.zylinder_sensoren[16].b_ausgefahren := zyl_haspel_re_abspulen.fb.e_sensor1_ausgefahren;


			BANDWECHSLER_V2:(*noch anpassen*)
				(* Die Seitenbezeichnungen (links, rechts) beziehen sich auf die Maschinenvorderseite *)
				(* Haspel Links Heben *)
				zyl_haspel_li_heben.fb.b_direkttaste_ausfahren := visu_hinten.out.zylinder_direkttasten[0].b_ausfahren;
				zyl_haspel_li_heben.fb.b_direkttaste_einfahren := visu_hinten.out.zylinder_direkttasten[0].b_einfahren;
				visu_hinten.in.zylinder_sensoren[0].b_eingefahren := NOT zyl_haspel_li_heben.fb.e_sensor1_ausgefahren;
				visu_hinten.in.zylinder_sensoren[0].b_ausgefahren := zyl_haspel_li_heben.fb.e_sensor1_ausgefahren;

				(* Haspel Links Sperren *)
				zyl_haspel_li_sperren.fb.b_direkttaste_ausfahren := visu_hinten.out.zylinder_direkttasten[1].b_ausfahren;
				zyl_haspel_li_sperren.fb.b_direkttaste_einfahren :=  visu_hinten.out.zylinder_direkttasten[1].b_einfahren;
				zyl_haspel_li_abspulen.fb.b_direkttaste_ausfahren:=visu_hinten.out.zylinder_direkttasten[1].b_einfahren; (*Abspulzylinder beim Entriegeln anheben*)
				visu_hinten.in.zylinder_sensoren[1].b_eingefahren := zyl_haspel_li_sperren.fb.e_sensor1_eingefahren;
				visu_hinten.in.zylinder_sensoren[1].b_ausgefahren := zyl_haspel_li_sperren.fb.e_sensor1_ausgefahren;

				(* Haspel Rechts Heben *)
				zyl_haspel_re_heben.fb.b_direkttaste_ausfahren := visu_hinten.out.zylinder_direkttasten[2].b_ausfahren;
				zyl_haspel_re_heben.fb.b_direkttaste_einfahren := visu_hinten.out.zylinder_direkttasten[2].b_einfahren;
				visu_hinten.in.zylinder_sensoren[2].b_eingefahren := NOT zyl_haspel_re_heben.fb.e_sensor1_ausgefahren;
				visu_hinten.in.zylinder_sensoren[2].b_ausgefahren := zyl_haspel_re_heben.fb.e_sensor1_ausgefahren;

				(* Haspel Rechts Sperren *)
				zyl_haspel_re_sperren.fb.b_direkttaste_ausfahren := visu_hinten.out.zylinder_direkttasten[3].b_ausfahren;
				zyl_haspel_re_sperren.fb.b_direkttaste_einfahren := visu_hinten.out.zylinder_direkttasten[3].b_einfahren;
				zyl_haspel_re_abspulen.fb.b_direkttaste_ausfahren:=visu_hinten.out.zylinder_direkttasten[3].b_einfahren; (*Abspulzylinder beim Entriegeln anheben*)
				visu_hinten.in.zylinder_sensoren[3].b_eingefahren := zyl_haspel_re_sperren.fb.e_sensor1_eingefahren;
				visu_hinten.in.zylinder_sensoren[3].b_ausgefahren := zyl_haspel_re_sperren.fb.e_sensor1_ausgefahren;

				(* Bandfänger *)
				zyl_bandfaenger.fb.b_direkttaste_ausfahren := visu_hinten.out.zylinder_direkttasten[4].b_ausfahren;
				zyl_bandfaenger.fb.b_direkttaste_einfahren := visu_hinten.out.zylinder_direkttasten[4].b_einfahren;
				visu_hinten.in.zylinder_sensoren[4].b_eingefahren := zyl_bandfaenger.fb.a_ventil_einfahren;
				visu_hinten.in.zylinder_sensoren[4].b_ausgefahren := zyl_bandfaenger.fb.a_ventil_ausfahren;
		
				(* Bandklemmen *)
				zyl_bandklemmen.fb.b_direkttaste_ausfahren := visu_hinten.out.zylinder_direkttasten[5].b_ausfahren;
				zyl_bandklemmen.fb.b_direkttaste_einfahren := visu_hinten.out.zylinder_direkttasten[5].b_einfahren;
				visu_hinten.in.zylinder_sensoren[5].b_eingefahren := zyl_bandklemmen.fb.a_ventil_einfahren;
				visu_hinten.in.zylinder_sensoren[5].b_ausgefahren := zyl_bandklemmen.fb.a_ventil_ausfahren;
		
				(* Bandwechselhalter links *)
				zyl_bawe_halter_li.fb.b_direkttaste_ausfahren := visu_hinten.out.zylinder_direkttasten[6].b_ausfahren;
				zyl_bawe_halter_li.fb.b_direkttaste_einfahren := visu_hinten.out.zylinder_direkttasten[6].b_einfahren;
				visu_hinten.in.zylinder_sensoren[6].b_eingefahren := zyl_bawe_halter_li.fb.a_ventil_einfahren;
				visu_hinten.in.zylinder_sensoren[6].b_ausgefahren := zyl_bawe_halter_li.fb.a_ventil_ausfahren;
		
				(* Bandwechselhalter rechts *)
				zyl_bawe_halter_re.fb.b_direkttaste_ausfahren := visu_hinten.out.zylinder_direkttasten[7].b_ausfahren;
				zyl_bawe_halter_re.fb.b_direkttaste_einfahren := visu_hinten.out.zylinder_direkttasten[7].b_einfahren;
				visu_hinten.in.zylinder_sensoren[7].b_eingefahren := zyl_bawe_halter_re.fb.a_ventil_einfahren;
				visu_hinten.in.zylinder_sensoren[7].b_ausgefahren := zyl_bawe_halter_re.fb.a_ventil_ausfahren;
		
				(* Bandwechselfänger links *)
				zyl_bawe_faenger_li.fb.b_direkttaste_ausfahren := visu_hinten.out.zylinder_direkttasten[8].b_ausfahren;
				zyl_bawe_faenger_li.fb.b_direkttaste_einfahren := visu_hinten.out.zylinder_direkttasten[8].b_einfahren;
				visu_hinten.in.zylinder_sensoren[8].b_eingefahren := zyl_bawe_faenger_li.fb.a_ventil_einfahren;
				visu_hinten.in.zylinder_sensoren[8].b_ausgefahren := zyl_bawe_faenger_li.fb.a_ventil_ausfahren;
		
				(* Bandwechselfänger rechts *)
				zyl_bawe_faenger_re.fb.b_direkttaste_ausfahren := visu_hinten.out.zylinder_direkttasten[9].b_ausfahren;
				zyl_bawe_faenger_re.fb.b_direkttaste_einfahren := visu_hinten.out.zylinder_direkttasten[9].b_einfahren;
				visu_hinten.in.zylinder_sensoren[9].b_eingefahren := zyl_bawe_faenger_re.fb.a_ventil_einfahren;
				visu_hinten.in.zylinder_sensoren[9].b_ausgefahren := zyl_bawe_faenger_re.fb.a_ventil_ausfahren;

				(*Spulenwechsel bie 1700======================*)
				(*Quervorschub*)
				zyl_bawe_querschub.st_ctrl.in.b_ausfahren := visu_hinten.out.zylinder_direkttasten[12].b_ausfahren;
				zyl_bawe_querschub.st_ctrl.in.b_einfahren := visu_hinten.out.zylinder_direkttasten[12].b_einfahren;

				visu_hinten.in.zylinder_sensoren[12].b_eingefahren := zyl_bawe_querschub.fb.e_sensor1_eingefahren;
				visu_hinten.in.zylinder_sensoren[12].b_ausgefahren := zyl_bawe_querschub.fb.e_sensor1_ausgefahren;

				(*Haspel verschieben*)
				zyl_haspel_verschieben.st_ctrl.in.b_ausfahren := visu_hinten.out.zylinder_direkttasten[13].b_ausfahren;
				zyl_haspel_verschieben.st_ctrl.in.b_einfahren := visu_hinten.out.zylinder_direkttasten[13].b_einfahren;

				visu_hinten.in.zylinder_sensoren[13].b_eingefahren := zyl_haspel_verschieben.fb.e_sensor1_eingefahren;
				visu_hinten.in.zylinder_sensoren[13].b_ausgefahren := zyl_haspel_verschieben.fb.e_sensor1_ausgefahren;

				(*Bandeinzug verschieben*)
				zyl_bandeinzuege_verschieben.st_ctrl.in.b_ausfahren := visu_hinten.out.zylinder_direkttasten[14].b_ausfahren;
				zyl_bandeinzuege_verschieben.st_ctrl.in.b_einfahren := visu_hinten.out.zylinder_direkttasten[14].b_einfahren;

				visu_hinten.in.zylinder_sensoren[14].b_eingefahren := zyl_bandeinzuege_verschieben.fb.e_sensor1_eingefahren;
				visu_hinten.in.zylinder_sensoren[14].b_ausgefahren := zyl_bandeinzuege_verschieben.fb.e_sensor1_ausgefahren;

				(* Haspel Links abspulen *)
				zyl_haspel_li_abspulen.fb.b_direkttaste_ausfahren := visu_hinten.out.zylinder_direkttasten[15].b_ausfahren;
				zyl_haspel_li_abspulen.fb.b_direkttaste_einfahren := visu_hinten.out.zylinder_direkttasten[15].b_einfahren;
				visu_hinten.in.zylinder_sensoren[15].b_eingefahren := NOT zyl_haspel_li_abspulen.fb.e_sensor1_ausgefahren;
				visu_hinten.in.zylinder_sensoren[15].b_ausgefahren := zyl_haspel_li_abspulen.fb.e_sensor1_ausgefahren;

				(* Haspel Rechts abspulen *)
				zyl_haspel_re_abspulen.fb.b_direkttaste_ausfahren := visu_hinten.out.zylinder_direkttasten[16].b_ausfahren;
				zyl_haspel_re_abspulen.fb.b_direkttaste_einfahren := visu_hinten.out.zylinder_direkttasten[16].b_einfahren;
				visu_hinten.in.zylinder_sensoren[16].b_eingefahren := NOT zyl_haspel_re_abspulen.fb.e_sensor1_ausgefahren;
				visu_hinten.in.zylinder_sensoren[16].b_ausgefahren := zyl_haspel_re_abspulen.fb.e_sensor1_ausgefahren;


		END_CASE

	BESTUECKZELLE_1720:

		CASE gst_datensatz.st_wkz.i16_typ_bandeinzug OF
			KEIN_EINZUG:
				;

			STANDARD_2FACH_V2:(*noch anpassen*)
				(* Die Seitenbezeichnungen (links, rechts) beziehen sich auf die Maschinenvorderseite *)
				(* Haspel Links Heben *)
				zyl_haspel_li_heben.fb.b_direkttaste_ausfahren := visu_hinten.out.zylinder_direkttasten[0].b_ausfahren;
				zyl_haspel_li_heben.fb.b_direkttaste_einfahren := visu_hinten.out.zylinder_direkttasten[0].b_einfahren;
				visu_hinten.in.zylinder_sensoren[0].b_eingefahren := zyl_haspel_li_heben.fb.a_ventil_einfahren;
				visu_hinten.in.zylinder_sensoren[0].b_ausgefahren := zyl_haspel_li_heben.fb.a_ventil_ausfahren;

				(* Haspel Links Sperren *)
				zyl_haspel_li_sperren.fb.b_direkttaste_ausfahren := visu_hinten.out.zylinder_direkttasten[1].b_ausfahren;
				zyl_haspel_li_sperren.fb.b_direkttaste_einfahren :=  visu_hinten.out.zylinder_direkttasten[1].b_einfahren;
				zyl_haspel_li_abspulen.fb.b_direkttaste_ausfahren:=visu_hinten.out.zylinder_direkttasten[1].b_einfahren; (*Abspulzylinder beim Entriegeln anheben*)
				visu_hinten.in.zylinder_sensoren[1].b_eingefahren := zyl_haspel_li_sperren.fb.a_ventil_einfahren;
				visu_hinten.in.zylinder_sensoren[1].b_ausgefahren := zyl_haspel_li_sperren.fb.a_ventil_ausfahren;

				(* Haspel Rechts Heben *)
				zyl_haspel_re_heben.fb.b_direkttaste_ausfahren := visu_hinten.out.zylinder_direkttasten[2].b_ausfahren;
				zyl_haspel_re_heben.fb.b_direkttaste_einfahren := visu_hinten.out.zylinder_direkttasten[2].b_einfahren;
				visu_hinten.in.zylinder_sensoren[2].b_eingefahren := zyl_haspel_re_heben.fb.a_ventil_einfahren;
				visu_hinten.in.zylinder_sensoren[2].b_ausgefahren := zyl_haspel_re_heben.fb.a_ventil_ausfahren;
		
				(* Haspel Rechts Sperren *)
				zyl_haspel_re_sperren.fb.b_direkttaste_ausfahren := visu_hinten.out.zylinder_direkttasten[3].b_ausfahren;
				zyl_haspel_re_sperren.fb.b_direkttaste_einfahren := visu_hinten.out.zylinder_direkttasten[3].b_einfahren;
				zyl_haspel_re_abspulen.fb.b_direkttaste_ausfahren:=visu_hinten.out.zylinder_direkttasten[3].b_einfahren; (*Abspulzylinder beim Entriegeln anheben*)
				visu_hinten.in.zylinder_sensoren[3].b_eingefahren := zyl_haspel_re_sperren.fb.a_ventil_einfahren;
				visu_hinten.in.zylinder_sensoren[3].b_ausgefahren := zyl_haspel_re_sperren.fb.a_ventil_ausfahren;
		
					(* Bandeinzug links: Bandfänger *)
				zyl_bandfaenger_li.fb.b_direkttaste_ausfahren := visu_hinten.out.zylinder_direkttasten[9].b_ausfahren;
				zyl_bandfaenger_li.fb.b_direkttaste_einfahren := visu_hinten.out.zylinder_direkttasten[9].b_einfahren;
				visu_hinten.in.zylinder_sensoren[9].b_eingefahren := zyl_bandfaenger_li.fb.a_ventil_einfahren;
				visu_hinten.in.zylinder_sensoren[9].b_ausgefahren := zyl_bandfaenger_li.fb.a_ventil_ausfahren;

				(* Bandeinzug links: Bandklemmen *)
				zyl_bandklemmen_li.fb.b_direkttaste_ausfahren := visu_hinten.out.zylinder_direkttasten[11].b_ausfahren;
				zyl_bandklemmen_li.fb.b_direkttaste_einfahren := visu_hinten.out.zylinder_direkttasten[11].b_einfahren;
				visu_hinten.in.zylinder_sensoren[11].b_eingefahren := zyl_bandklemmen_li.fb.a_ventil_einfahren;
				visu_hinten.in.zylinder_sensoren[11].b_ausgefahren := zyl_bandklemmen_li.fb.a_ventil_ausfahren;
		
				(* Bandeinzug rechts: Bandfänger *)
				zyl_bandfaenger_re.fb.b_direkttaste_ausfahren := visu_hinten.out.zylinder_direkttasten[8].b_ausfahren;
				zyl_bandfaenger_re.fb.b_direkttaste_einfahren := visu_hinten.out.zylinder_direkttasten[8].b_einfahren;
				visu_hinten.in.zylinder_sensoren[8].b_eingefahren := zyl_bandfaenger_re.fb.a_ventil_einfahren;
				visu_hinten.in.zylinder_sensoren[8].b_ausgefahren := zyl_bandfaenger_re.fb.a_ventil_ausfahren;
		
				(* Bandeinzug rechts: Bandklemmen *)
				zyl_bandklemmen_re.fb.b_direkttaste_ausfahren := visu_hinten.out.zylinder_direkttasten[10].b_ausfahren;
				zyl_bandklemmen_re.fb.b_direkttaste_einfahren := visu_hinten.out.zylinder_direkttasten[10].b_einfahren;
				visu_hinten.in.zylinder_sensoren[10].b_eingefahren := zyl_bandklemmen_re.fb.a_ventil_einfahren;
				visu_hinten.in.zylinder_sensoren[10].b_ausgefahren := zyl_bandklemmen_re.fb.a_ventil_ausfahren;

				(* Bandwechselhalter links *)
				zyl_bawe_halter_li.fb.b_direkttaste_ausfahren := visu_hinten.out.zylinder_direkttasten[7].b_ausfahren;
				zyl_bawe_halter_li.fb.b_direkttaste_einfahren := visu_hinten.out.zylinder_direkttasten[7].b_einfahren;
				visu_hinten.in.zylinder_sensoren[7].b_eingefahren := zyl_bawe_halter_li.fb.e_sensor1_eingefahren;
				visu_hinten.in.zylinder_sensoren[7].b_ausgefahren := zyl_bawe_halter_li.fb.e_sensor1_ausgefahren;
		
				(* Bandwechselhalter rechts *)
				zyl_bawe_halter_re.fb.b_direkttaste_ausfahren := visu_hinten.out.zylinder_direkttasten[6].b_ausfahren;
				zyl_bawe_halter_re.fb.b_direkttaste_einfahren := visu_hinten.out.zylinder_direkttasten[6].b_einfahren;
				visu_hinten.in.zylinder_sensoren[6].b_eingefahren := zyl_bawe_halter_re.fb.e_sensor1_eingefahren;
				visu_hinten.in.zylinder_sensoren[6].b_ausgefahren := zyl_bawe_halter_re.fb.e_sensor1_ausgefahren;

				(* Haspel Links abspulen *)
				zyl_haspel_li_abspulen.fb.b_direkttaste_ausfahren := visu_hinten.out.zylinder_direkttasten[15].b_ausfahren;
				zyl_haspel_li_abspulen.fb.b_direkttaste_einfahren := visu_hinten.out.zylinder_direkttasten[15].b_einfahren;
				visu_hinten.in.zylinder_sensoren[15].b_eingefahren := NOT zyl_haspel_li_abspulen.fb.e_sensor1_ausgefahren;
				visu_hinten.in.zylinder_sensoren[15].b_ausgefahren := zyl_haspel_li_abspulen.fb.e_sensor1_ausgefahren;

				(* Haspel Rechts abspulen *)
				zyl_haspel_re_abspulen.fb.b_direkttaste_ausfahren := visu_hinten.out.zylinder_direkttasten[16].b_ausfahren;
				zyl_haspel_re_abspulen.fb.b_direkttaste_einfahren := visu_hinten.out.zylinder_direkttasten[16].b_einfahren;
				visu_hinten.in.zylinder_sensoren[16].b_eingefahren := NOT zyl_haspel_re_abspulen.fb.e_sensor1_ausgefahren;
				visu_hinten.in.zylinder_sensoren[16].b_ausgefahren := zyl_haspel_re_abspulen.fb.e_sensor1_ausgefahren;

			BANDWECHSLER_V2:
				;

			SERVO:
				;
		END_CASE




	RASTERFOLIE:
		(* Die Seitenbezeichnungen (links, rechts) beziehen sich auf die Maschinenvorderseite *)
		(* Haspel Links Heben *)
		zyl_haspel_li_heben.fb.b_direkttaste_ausfahren := visu_hinten.out.zylinder_direkttasten[0].b_ausfahren;
		zyl_haspel_li_heben.fb.b_direkttaste_einfahren := visu_hinten.out.zylinder_direkttasten[0].b_einfahren;
		visu_hinten.in.zylinder_sensoren[0].b_eingefahren := zyl_haspel_li_heben.fb.e_sensor1_eingefahren;
		visu_hinten.in.zylinder_sensoren[0].b_ausgefahren := zyl_haspel_li_heben.fb.e_sensor1_ausgefahren;

		(* Haspel Links Sperren *)
		zyl_haspel_li_sperren.fb.b_direkttaste_ausfahren := visu_hinten.out.zylinder_direkttasten[1].b_ausfahren;
		zyl_haspel_li_sperren.fb.b_direkttaste_einfahren :=  visu_hinten.out.zylinder_direkttasten[1].b_einfahren;
		zyl_haspel_li_abspulen.fb.b_direkttaste_ausfahren:=visu_hinten.out.zylinder_direkttasten[1].b_einfahren; (*Abspulzylinder beim Entriegeln anheben*)
		visu_hinten.in.zylinder_sensoren[1].b_eingefahren := zyl_haspel_li_sperren.fb.e_sensor1_eingefahren;
		visu_hinten.in.zylinder_sensoren[1].b_ausgefahren := zyl_haspel_li_sperren.fb.e_sensor1_ausgefahren;

		(* Haspel Rechts Heben *)
		zyl_haspel_re_heben.fb.b_direkttaste_ausfahren := visu_hinten.out.zylinder_direkttasten[2].b_ausfahren;
		zyl_haspel_re_heben.fb.b_direkttaste_einfahren := visu_hinten.out.zylinder_direkttasten[2].b_einfahren;
		visu_hinten.in.zylinder_sensoren[2].b_eingefahren := zyl_haspel_re_heben.fb.e_sensor1_eingefahren;
		visu_hinten.in.zylinder_sensoren[2].b_ausgefahren := zyl_haspel_re_heben.fb.e_sensor1_ausgefahren;

		(* Haspel Rechts Sperren *)
		zyl_haspel_re_sperren.fb.b_direkttaste_ausfahren := visu_hinten.out.zylinder_direkttasten[3].b_ausfahren;
		zyl_haspel_re_sperren.fb.b_direkttaste_einfahren := visu_hinten.out.zylinder_direkttasten[3].b_einfahren;
		zyl_haspel_re_abspulen.fb.b_direkttaste_ausfahren:=visu_hinten.out.zylinder_direkttasten[3].b_einfahren; (*Abspulzylinder beim Entriegeln anheben*)
		visu_hinten.in.zylinder_sensoren[3].b_eingefahren := zyl_haspel_re_sperren.fb.e_sensor1_eingefahren;
		visu_hinten.in.zylinder_sensoren[3].b_ausgefahren := zyl_haspel_re_sperren.fb.e_sensor1_ausgefahren;

		(* Folienfänger *)
		zyl_rafo_faenger.fb.b_direkttaste_ausfahren := visu_hinten.out.zylinder_direkttasten[4].b_ausfahren;
		zyl_rafo_faenger.fb.b_direkttaste_einfahren := visu_hinten.out.zylinder_direkttasten[4].b_einfahren;
		visu_hinten.in.zylinder_sensoren[4].b_eingefahren := zyl_rafo_faenger.fb.e_sensor1_eingefahren;
		visu_hinten.in.zylinder_sensoren[4].b_ausgefahren := zyl_rafo_faenger.fb.e_sensor1_ausgefahren;

		(* Folienklemmen *)
		zyl_rafo_klemmen.fb.b_direkttaste_ausfahren := visu_hinten.out.zylinder_direkttasten[5].b_ausfahren;
		zyl_rafo_klemmen.fb.b_direkttaste_einfahren := visu_hinten.out.zylinder_direkttasten[5].b_einfahren;
		visu_hinten.in.zylinder_sensoren[5].b_eingefahren := zyl_rafo_klemmen.fb.e_sensor1_eingefahren;
		visu_hinten.in.zylinder_sensoren[5].b_ausgefahren := zyl_rafo_klemmen.fb.e_sensor1_ausgefahren;
END_CASE
END_PROGRAM

(* POU Gemeinsamkeiten17xx/Wartung/ST_Wartung, ST *)
PROGRAM ST_Wartung
VAR_INPUT
	st_config								: struct_config;
	st_ctrl_in								: struct_ctrl_in;
END_VAR
VAR_IN_OUT
	i16_auftrag							: enum_wartung_auftrag;
END_VAR
VAR_OUTPUT
	st_ctrl_out								: struct_ctrl_out;
END_VAR
VAR
	(*Bausteinaufrufe*)
	fb_state_entry					: ST_StateEntry;
	fb_ton_quitt						: TON;
	fb_xml_srv_read					: FB_XmlSrvReadByName;
	fb_xml_srv_write					: FB_XmlSrvWriteByName;
	fbFindFiles						: FB_EnumFindFileList;
	file								: ST_FindFileEntry;
	FB_GetHostName				: FB_GetHostName;
	fb_nt_start_process				: NT_StartProcess;

	(*Flanken*)
	fb_r_trig_autosafe				: R_TRIG;
	fb_r_trig_reset_wkz			: R_TRIG;

	(*Zeiten*)
	fb_ton_wz									: TON;
	fb_ton_wz_wartung				: TON;
	fb_ton_end								: TON;
	fb_ton_autosafe					: TON;


	(* Dateiname *)
	sFileName_md							: STRING;
	sFileName_wkz						: STRING;
	sHelpName							: STRING;
	sHelpPos							: INT;

	(* Dateipfad *)
	sPathName								: STRING;

	(* Temporäre Variable *)
	b_init											: BOOL;
	b_lesen_komplett					: BOOL := TRUE;
	b_datei_vorhanden				: BOOL;
	b_auto_speichern_auf_server		: BOOL ;
	nErrId											: UDINT;
	sm_fehler_schreiben_Wartungsprotokoll			: BOOL;
	sm_fehler_lesen_Wartungsprotokoll					: BOOL;
	sm_fehler_speichern_Wartungsprotokoll			: BOOL;

	s_aktuelles_wkz_copy											: STRING;
	i																					: INT:=0;

	st_wartungsprotokoll_md_copy							: struct_Wartungsprotokoll;
	st_wartungsprotokoll_wkz_copy							: struct_Wartungsprotokoll;
	i32_bestueckhubzaehler_md_copy					: UDINT := 0;
	i32_bestueckhubzaehler_wkz_copy				: UDINT := 0;
END_VAR

VAR CONSTANT
	st_wartungsprotokoll_leer			: struct_Wartungsprotokoll;
	s_wartung_path_wkz					: STRING(50):='D:\BBgen\Wartung\Werkzeug\';
	s_wartung_path_md						: STRING(50):='D:\BBgen\Wartung\Maschine\';
	s_Trennstelle									: STRING(2):='#';
END_VAR
FileName_erstellen ();
fb_Aufrufe ();
auto_speichern_laden ();

IF NOT b_init AND gst_datensatz.st_md.s_aktuelles_wkz <>''  THEN
	i16_auftrag:= LESE_WARTUNGSPROTOKOLL_KOMPLETT;
	s_aktuelles_wkz_copy:=gst_datensatz.st_md.s_aktuelles_wkz;
	i32_bestueckhubzaehler_md_copy:=gst_datensatz.st_md.i32_bestueckhubzaehler;
	FB_GetHostName.bExecute := TRUE;
	b_init := TRUE;
ELSIF b_init AND gst_datensatz.st_md.s_aktuelles_wkz <> s_aktuelles_wkz_copy AND gi16_maschinenstatusinfo <> STATUS_MASCHINE_ARBEITET THEN
	i16_auftrag:=LESE_WARTUNGSPROTOKOLL_WKZ;
	i32_bestueckhubzaehler_md_copy:=gst_datensatz.st_md.i32_bestueckhubzaehler;
	s_aktuelles_wkz_copy:=gst_datensatz.st_md.s_aktuelles_wkz;
ELSE
	Zaehler();
END_IF


(*Zellennummer aus dem Computernamen filtern*)
sHelpName := FB_GetHostName.sHostName;
sHelpPos := FIND(sHelpName,'-');
sHelpName := DELETE(sHelpName,sHelpPos,1);
sHelpPos := FIND(sHelpName,'-');
sHelpName := LEFT(sHelpName,sHelpPos-1);
sHelpName := CONCAT('T#',sHelpName);
sHelpName := CONCAT(sHelpName,'s');

(* Flanken *)
fb_r_trig_reset_wkz(CLK:= visu.b_reset_wartung_wkz, Q=> );
fb_r_trig_autosafe(CLK:= gstr_uhrzeit = '01:00:00', Q=> );
fb_ton_autosafe(IN:= , PT:= STRING_TO_TIME(sHelpName), Q=> , ET=> );

IF fb_r_trig_autosafe.Q THEN
	fb_ton_autosafe.IN := TRUE;
END_IF

(*Um 1 Uhr + Zellennummer in Sek. früh werden die Wartungsprotokolle an den Server geschickt*)
IF fb_ton_autosafe.Q THEN
	b_auto_speichern_auf_server := TRUE;
	fb_ton_autosafe.IN := FALSE;
END_IF

IF b_auto_speichern_auf_server AND i16_auftrag = KEIN_WARTUNG_AUFTRAG THEN
	b_auto_speichern_auf_server := FALSE;
	IF visu.s_akt_sprache = 'de' THEN
		i16_auftrag:=SPEICHERN_WARTUNGSPROTOKOLL;
	END_IF
END_IF


(*
IF visu.b_reset_wartung_maschine THEN
	gst_datensatz.st_md.produzierte_stecker := 0;
END_IF
*)

(*Zeiten*)
fb_ton_wz(IN:= , PT:= , Q=> , ET=> );
fb_ton_quitt(IN:= , PT:= t#100ms, Q=> , ET=> );

(* ======================================Schrittkette======================================== *)
fb_state_entry(i16_pos:= 1);


CASE fb_state_entry.i16_step OF
(*=======================================================*)
	INIT_OBJ:
		(*-----------------------Weiterschaltbedingungen----------------------------*)
		IF FB_GetHostName.bBusy OR FB_GetHostName.sHostName <> '' THEN
			fb_state_entry.i16_next_step := 5;
		END_IF

		IF fb_state_entry.X THEN
			FB_GetHostName.bExecute := FALSE;
		END_IF

(*=======================================================*)
	5:
		(*-----------------------Weiterschaltbedingungen----------------------------*)
		IF NOT FB_GetHostName.bBusy THEN
			fb_state_entry.i16_next_step := INIT;
		END_IF

(*=======================================================*)
	INIT:	(*initialisieren*)
		st_ctrl_out.b_fehler := FALSE;
		st_ctrl_out.b_bereit := FALSE;
		st_ctrl_out.b_busy := FALSE;
		st_ctrl_out.b_fertig := FALSE;
		sm_fehler_schreiben_Wartungsprotokoll	 := FALSE;
		sm_fehler_lesen_Wartungsprotokoll	:= FALSE;
		sm_fehler_speichern_Wartungsprotokoll := FALSE;
		fbFindFiles.bExecute := FALSE;
		fb_xml_srv_write.bExecute := FALSE;
		fb_xml_srv_read.bExecute := FALSE;
		fb_ton_wz.IN := FALSE;

		fb_nt_start_process.START := FALSE;
		fbFindFiles.eCmd := 0;
		nErrId := 0;
		sPathName := '';
		b_datei_vorhanden := FALSE;
		fb_xml_srv_write.sSymName := '';
		fb_xml_srv_write.sXPath := '';

		(*-----------------------Weiterschaltbedingungen----------------------------*)
		fb_state_entry.i16_next_step:=BEREIT;


(*=======================================================*)
	BEREIT:(*Start*)
		IF 	fb_state_entry.E THEN
			st_ctrl_out.b_bereit := TRUE;
		END_IF

		CASE i16_auftrag OF
			LESE_WARTUNGSPROTOKOLL_KOMPLETT:
				b_lesen_komplett := TRUE;
				fb_state_entry.i16_next_step:=110;

			LESE_WARTUNGSPROTOKOLL_WKZ:
				fb_state_entry.i16_next_step:=110;

			LESE_WARTUNGSPROTOKOLL_MD:
				fb_state_entry.i16_next_step:=150;

			SCHREIBE_WARTUNGSPROTOKOLL_WKZ:
				fb_state_entry.i16_next_step:=200;

			SCHREIBE_WARTUNGSPROTOKOLL_MD:
				fb_state_entry.i16_next_step:=250;

			SPEICHERN_WARTUNGSPROTOKOLL:
				fb_state_entry.i16_next_step:=300;

			SCHREIBE_WARTUNGSPROTOKOLL_WKZ_RESET:
				fb_state_entry.i16_next_step:=400;
		END_CASE

		IF fb_state_entry.X THEN
			st_ctrl_out.b_bereit := FALSE;
			st_ctrl_out.b_fertig := FALSE;
			st_ctrl_out.b_busy := TRUE;
		END_IF

(*=======================================================*)
	110:(*Prüfe, ob Werkzeug Datei vorhanden ist*)
		IF fb_state_entry.E THEN
			sPathName := CONCAT(s_wartung_path_wkz,sFileName_wkz);
			sPathName:=CONCAT(sPathName,'.xml');
			(*Erste Datei im Verzeichnis kontrollieren*)
			IF fb_state_entry.i16_last_step <> 120 THEN
				fbFindFiles.eCmd := 0;
			(*Dateien im Verzeichnis durchzählen*)
			ELSE
				fbFindFiles.eCmd := 1;
			END_IF
			fbFindFiles.bExecute := TRUE;
		END_IF

		(*-----------------------Weiterschaltbedingungen----------------------------*)
		IF fbFindFiles.bBusy THEN
			fb_state_entry.i16_next_step:=120;
		END_IF

		IF fb_state_entry.X THEN
			fbFindFiles.bExecute := FALSE;
		END_IF

(*=======================================================*)
	120:(*Prüfe, ob Werkzeug Datei vorhanden ist*)
		(*-----------------------Weiterschaltbedingungen----------------------------*)
		(*letzte Datei im Verzeichnis erreicht*)
		IF fbFindFiles.bEOE AND NOT fbFindFiles.bBusy AND NOT fbFindFiles.bError  THEN
			IF fbFindFiles.nFindFiles <> 0 OR b_datei_vorhanden  THEN
				(*Datei vorhanden -> muss eingelesen werden*)
				fb_state_entry.i16_next_step:=130;
			ELSE
				(*Datei noch nicht vorhanden -> kann nicht eingelesen werden*)
				i32_bestueckhubzaehler_wkz_copy := 0;
				IF b_lesen_komplett THEN
					fb_state_entry.i16_next_step:=150;
				ELSE
					fb_state_entry.i16_next_step := 999;
				END_IF
			END_IF
		(*Datei wurde im Verzeichnis gefunden*)
		ELSIF NOT fbFindFiles.bBusy AND NOT fbFindFiles.bError  THEN
			IF fbFindFiles.nFindFiles <> 0  THEN
				(*Datei vorhanden -> muss eingelesen werden*)
				b_datei_vorhanden := TRUE;
				fb_state_entry.i16_next_step := 110;
			END_IF
		ELSIF fbFindFiles.bError THEN
			nErrId := fbFindFiles.nErrID;
			sm_fehler_lesen_Wartungsprotokoll := TRUE;
			fb_state_entry.i16_next_step:=FEHLER;
		END_IF

(*=======================================================*)
	130:	(* Lesen Werkzeug Wartungsprotokoll *)
		IF fb_state_entry.E THEN
			b_datei_vorhanden := FALSE;
			sPathName := CONCAT(s_wartung_path_wkz,sFileName_wkz);
			sPathName:=CONCAT(sPathName,'.xml');
			fb_xml_srv_read.sSymName := '.gst_datensatz.st_wartungsprotokoll.st_wartung_wkz';
			fb_xml_srv_read.sXPath := '/root/gst_datensatz.st_wartungsprotokoll.st_wartung_wkz';
			fb_xml_srv_read.bExecute:= TRUE;
		END_IF

		(*-----------------------Weiterschaltbedingungen----------------------------*)
		IF fb_xml_srv_read.bBusy THEN
			fb_state_entry.i16_next_step := 140;
		END_IF

		IF fb_state_entry.X THEN
			fb_xml_srv_read.bExecute:= FALSE;
		END_IF

(*=======================================================*)
	140:
		(*-----------------------Weiterschaltbedingungen----------------------------*)
		(*Lesen erfolgreich*)
		IF NOT fb_xml_srv_read.bError AND NOT fb_xml_srv_read.bBusy AND NOT b_lesen_komplett THEN
			i32_bestueckhubzaehler_wkz_copy := gst_datensatz.st_wartungsprotokoll.st_wartung_wkz.hubzaehler;
			fb_state_entry.i16_next_step := 999;
		ELSIF NOT fb_xml_srv_read.bError AND NOT fb_xml_srv_read.bBusy AND b_lesen_komplett THEN
			i32_bestueckhubzaehler_wkz_copy := gst_datensatz.st_wartungsprotokoll.st_wartung_wkz.hubzaehler;
			fb_state_entry.i16_next_step := 150;
		ELSIF fb_xml_srv_read.bError THEN
			nErrId:=fb_xml_srv_read.nErrId;
			sm_fehler_lesen_Wartungsprotokoll:=TRUE;
			fb_state_entry.i16_next_step := FEHLER;
		END_IF

(*=======================================================*)
	150:(*Prüfe, ob Maschinen Datei vorhanden ist*)
		IF fb_state_entry.E THEN
			sPathName := CONCAT(s_wartung_path_md,sFileName_md);
			(*Erste Datei im Verzeichnis kontrollieren*)
			IF fb_state_entry.i16_last_step <> 160 THEN
				fbFindFiles.eCmd := 0;
			(*Dateien im Verzeichnis durchzählen*)
			ELSE
				fbFindFiles.eCmd := 1;
			END_IF
			fbFindFiles.bExecute := TRUE;
		END_IF

		(*-----------------------Weiterschaltbedingungen----------------------------*)
		IF fbFindFiles.bBusy THEN
			fb_state_entry.i16_next_step:=160;
		END_IF

		IF fb_state_entry.X THEN
			fbFindFiles.bExecute := FALSE;
		END_IF

(*=======================================================*)
	160:(*Prüfe, ob Maschinen Datei vorhanden ist*)
		(*-----------------------Weiterschaltbedingungen----------------------------*)
		(*letzte Datei im Verzeichnis erreicht*)
		IF fbFindFiles.bEOE AND NOT fbFindFiles.bBusy AND NOT fbFindFiles.bError  THEN
			IF fbFindFiles.nFindFiles <> 0 OR b_datei_vorhanden  THEN
				(*Datei vorhanden -> muss eingelesen werden*)
				fb_state_entry.i16_next_step:=170;
			ELSE
				(*Datei noch nicht vorhanden -> kann nicht eingelesen werden*)
				fb_state_entry.i16_next_step:=999;
			END_IF
		(*Datei wurde im Verzeichnis gefunden*)
		ELSIF NOT fbFindFiles.bBusy AND NOT fbFindFiles.bError  THEN
			IF fbFindFiles.nFindFiles <> 0  THEN
				(*Datei vorhanden -> muss eingelesen werden*)
				b_datei_vorhanden := TRUE;
				fb_state_entry.i16_next_step := 150;
			END_IF
		ELSIF fbFindFiles.bError THEN
			nErrId := fbFindFiles.nErrID;
			sm_fehler_lesen_wartungsprotokoll := TRUE;
			fb_state_entry.i16_next_step:=FEHLER;
		END_IF

		IF fb_state_entry.X THEN
			b_lesen_komplett := FALSE;
		END_IF

(*=======================================================*)
	170:	(* Lesen Maschinen Wartungsprotokoll *)
		IF fb_state_entry.E THEN
			b_datei_vorhanden := FALSE;
			sPathName := CONCAT(s_wartung_path_md,sFileName_md);
			fb_xml_srv_read.sSymName := '.gst_datensatz.st_wartungsprotokoll.st_wartung_md';
			fb_xml_srv_read.sXPath := '/root/gst_datensatz.st_wartungsprotokoll.st_wartung_md';
			fb_xml_srv_read.bExecute:= TRUE;
		END_IF

		(*-----------------------Weiterschaltbedingungen----------------------------*)
		IF fb_xml_srv_read.bBusy THEN
			fb_state_entry.i16_next_step := 180;
		END_IF

		IF fb_state_entry.X THEN
			fb_xml_srv_read.bExecute:= FALSE;
		END_IF

(*=======================================================*)
	180:
		(*-----------------------Weiterschaltbedingungen----------------------------*)
		(*Lesen erfolgreich*)
		IF NOT fb_xml_srv_read.bError AND NOT fb_xml_srv_read.bBusy THEN
			fb_state_entry.i16_next_step := 999;
		ELSIF fb_xml_srv_read.bError THEN
			nErrId:=fb_xml_srv_read.nErrId;
			sm_fehler_lesen_Wartungsprotokoll:=TRUE;
			fb_state_entry.i16_next_step := FEHLER;
		END_IF

(*=======================================================*)
	200:(*Schreibe Werkzeug Wartungsdatei*)
		IF fb_state_entry.E THEN
			sPathName := CONCAT(s_wartung_path_wkz,sFileName_wkz);
			sPathName:=CONCAT(sPathName,'.xml');
			fb_xml_srv_write.sSymName := '.gst_datensatz.st_wartungsprotokoll.st_wartung_wkz';
			fb_xml_srv_write.sXPath := '/root/gst_datensatz.st_wartungsprotokoll.st_wartung_wkz';
			fb_xml_srv_write.bExecute:= TRUE;
		END_IF

		(*-----------------------Weiterschaltbedingungen----------------------------*)
		IF fb_xml_srv_write.bBusy THEN
			fb_state_entry.i16_next_step := 210;
		END_IF

		IF fb_state_entry.X THEN
			fb_xml_srv_write.bExecute:= FALSE;
		END_IF

(*=======================================================*)
	210:
		(*-----------------------Weiterschaltbedingungen----------------------------*)
		IF NOT fb_xml_srv_write.bError AND NOT fb_xml_srv_write.bBusy THEN
			st_wartungsprotokoll_wkz_copy.st_wartung_wkz:= gst_datensatz.st_wartungsprotokoll.st_wartung_wkz ;
			fb_state_entry.i16_next_step := 999;
		END_IF


		IF fb_xml_srv_write.bError  THEN
			nErrId:=fb_xml_srv_write.nErrId;
			sm_fehler_schreiben_Wartungsprotokoll:=TRUE;
			fb_state_entry.i16_next_step := FEHLER;
		END_IF


(*===================Schrittkette====================================*)
	250:(*Schreibe Maschinen Wartungsdatei*)
		IF fb_state_entry.E THEN
			sPathName := CONCAT(s_wartung_path_md,sFileName_md);
			fb_xml_srv_write.sSymName := '.gst_datensatz.st_wartungsprotokoll.st_wartung_md';
			fb_xml_srv_write.sXPath := '/root/gst_datensatz.st_wartungsprotokoll.st_wartung_md';
			fb_xml_srv_write.bExecute:= TRUE;
		END_IF

		(*-----------------------Weiterschaltbedingungen----------------------------*)
		IF fb_xml_srv_write.bBusy THEN
			fb_state_entry.i16_next_step := 260;
		END_IF

		IF fb_state_entry.X THEN
			fb_xml_srv_write.bExecute:= FALSE;
		END_IF

(*=======================================================*)
	260:
		(*-----------------------Weiterschaltbedingungen----------------------------*)
		IF NOT fb_xml_srv_write.bError AND NOT fb_xml_srv_write.bBusy THEN
			st_wartungsprotokoll_md_copy.st_wartung_md:= gst_datensatz.st_wartungsprotokoll.st_wartung_md ;
			fb_state_entry.i16_next_step := 999;
		END_IF

		IF fb_xml_srv_write.bError  THEN
			nErrId:=fb_xml_srv_write.nErrId;
			sm_fehler_schreiben_Wartungsprotokoll:=TRUE;
			fb_state_entry.i16_next_step := FEHLER;
		END_IF

(*=======================================================*)
	300:(*Speichern der Wartungsdateien auf den Server*)
		IF 	fb_state_entry.E THEN
			fb_nt_start_process.START:=TRUE;
		END_IF

		IF fb_nt_start_process.BUSY THEN
			fb_state_entry.i16_next_step := 310;
			fb_nt_start_process.START:=FALSE;
		END_IF

(*=======================================================*)
	310:
		(*-----------------------Weiterschaltbedingungen----------------------------*)
		IF NOT fb_nt_start_process.ERR AND NOT fb_nt_start_process.BUSY THEN
			fb_state_entry.i16_next_step := 999;
		END_IF

		IF fb_nt_start_process.ERR THEN
			nErrId:=fb_nt_start_process.ERRID;
			sm_fehler_speichern_Wartungsprotokoll;
			fb_state_entry.i16_next_step:=FEHLER;
		END_IF

(*=======================================================*)
	400:(*Prüfe, ob Werkzeug Datei vorhanden ist*)
		IF fb_state_entry.E THEN
			sPathName := CONCAT(s_wartung_path_wkz,sFileName_wkz);
			sPathName:=CONCAT(sPathName,'_RESET');
			sPathName:=CONCAT(sPathName,'.xml');
			(*Erste Datei im Verzeichnis kontrollieren*)
			IF fb_state_entry.i16_last_step <> 410 THEN
				fbFindFiles.eCmd := 0;
			(*Dateien im Verzeichnis durchzählen*)
			ELSE
				fbFindFiles.eCmd := 1;
			END_IF
			fbFindFiles.bExecute := TRUE;
		END_IF

		(*-----------------------Weiterschaltbedingungen----------------------------*)
		IF fbFindFiles.bBusy THEN
			fb_state_entry.i16_next_step:=410;
		END_IF

		IF fb_state_entry.X THEN
			fbFindFiles.bExecute := FALSE;
		END_IF

(*=======================================================*)
	410:(*Prüfe, ob Werkzeug Datei vorhanden ist*)
		(*-----------------------Weiterschaltbedingungen----------------------------*)
		(*letzte Datei im Verzeichnis erreicht*)
		IF fbFindFiles.bEOE AND NOT fbFindFiles.bBusy AND NOT fbFindFiles.bError  THEN
			IF fbFindFiles.nFindFiles <> 0 OR b_datei_vorhanden  THEN
				(*Datei vorhanden -> darf nicht neu geschrieben werden*)
				fb_state_entry.i16_next_step:=999;
			ELSE
				(*Datei noch nicht vorhanden -> muss erstellt werden*)
				fb_state_entry.i16_next_step := 420;
			END_IF
		(*Datei wurde im Verzeichnis gefunden*)
		ELSIF NOT fbFindFiles.bBusy AND NOT fbFindFiles.bError  THEN
			IF fbFindFiles.nFindFiles <> 0  THEN
				(*Datei vorhanden -> muss eingelesen werden*)
				b_datei_vorhanden := TRUE;
				fb_state_entry.i16_next_step := 400;
			END_IF
		ELSIF fbFindFiles.bError THEN
			nErrId := fbFindFiles.nErrID;
			sm_fehler_lesen_Wartungsprotokoll := TRUE;
			fb_state_entry.i16_next_step:=FEHLER;
		END_IF

(*=======================================================*)
	420:(*Schreibe Werkzeug Reset Wartungsdatei*)
		IF fb_state_entry.E THEN
			sPathName := CONCAT(s_wartung_path_wkz,sFileName_wkz);
			sPathName:=CONCAT(sPathName,'_RESET');
			sPathName:=CONCAT(sPathName,'.xml');
			fb_xml_srv_write.sSymName := '.gst_datensatz.st_wartungsprotokoll.st_wartung_wkz';
			fb_xml_srv_write.sXPath := '/root/gst_datensatz.st_wartungsprotokoll.st_wartung_wkz';
			fb_xml_srv_write.bExecute:= TRUE;
		END_IF

		(*-----------------------Weiterschaltbedingungen----------------------------*)
		IF fb_xml_srv_write.bBusy THEN
			fb_state_entry.i16_next_step := 430;
		END_IF

		IF fb_state_entry.X THEN
			fb_xml_srv_write.bExecute:= FALSE;
		END_IF

(*=======================================================*)
	430:
		(*-----------------------Weiterschaltbedingungen----------------------------*)
		IF NOT fb_xml_srv_write.bError AND NOT fb_xml_srv_write.bBusy THEN
			i32_bestueckhubzaehler_md_copy:=gst_datensatz.st_md.i32_bestueckhubzaehler;
			s_aktuelles_wkz_copy:=gst_datensatz.st_md.s_aktuelles_wkz;
			gst_datensatz.st_wartungsprotokoll.st_wartung_wkz.hubzaehler := 0;
			i32_bestueckhubzaehler_wkz_copy := 0;
			fb_state_entry.i16_next_step := 999;
		END_IF

		IF fb_xml_srv_write.bError  THEN
			nErrId:=fb_xml_srv_write.nErrId;
			sm_fehler_schreiben_Wartungsprotokoll:=TRUE;
			fb_state_entry.i16_next_step := FEHLER;
		END_IF


(*=======================================================*)
	999:	(* Ende - Befehl wurde korrekt abgearbeitet *)
		IF fb_state_entry.E THEN
			b_datei_vorhanden := FALSE;
			st_ctrl_out.b_busy := FALSE;
			st_ctrl_out.b_fertig := TRUE;
			i16_auftrag := KEIN_WARTUNG_AUFTRAG;
			fb_state_entry.i16_next_step := BEREIT;
		END_IF

(*=======================================================*)
	FEHLER: (* Fehler *)
		IF fb_state_entry.E THEN
			i16_auftrag := KEIN_WARTUNG_AUFTRAG;
			st_ctrl_out.b_bereit := FALSE;
			st_ctrl_out.b_busy := FALSE;
			st_ctrl_out.b_fertig := FALSE;
			st_ctrl_out.b_fehler := TRUE;
			fb_ton_quitt.IN := FALSE;
		END_IF

		(*-----------------------Weiterschaltbedingungen----------------------------*)
		IF st_ctrl_in.b_quitt AND NOT fb_state_entry.E THEN
			st_ctrl_out.b_fehler := FALSE;
			fb_ton_quitt.IN := TRUE;
		END_IF

		IF fb_ton_quitt.Q THEN
			fb_ton_quitt.IN := FALSE;
			fb_state_entry.i16_next_step := INIT;
		END_IF
END_CASE

fb_state_entry(i16_pos:= 2 );

(* ======================================Subkomponenten======================================== *)

IF st_config.b_config_fertig THEN
	garr_stoermeldungen[st_config.i16_meld_startindex + 0] := sm_fehler_schreiben_Wartungsprotokoll;
	garr_stoermeldungen[st_config.i16_meld_startindex + 1] := sm_fehler_lesen_Wartungsprotokoll;
	garr_stoermeldungen[st_config.i16_meld_startindex + 2] := sm_fehler_speichern_Wartungsprotokoll;
	garr_stoermeldungen[st_config.i16_meld_startindex + 3] := FALSE;
	garr_stoermeldungen[st_config.i16_meld_startindex + 4] := FALSE;
	garr_stoermeldungen[st_config.i16_meld_startindex + 5] := FALSE;
	garr_stoermeldungen[st_config.i16_meld_startindex + 6] := FALSE;
	garr_stoermeldungen[st_config.i16_meld_startindex + 7] := FALSE;
	garr_stoermeldungen[st_config.i16_meld_startindex + 8] := FALSE;
	garr_stoermeldungen[st_config.i16_meld_startindex + 9] := FALSE;
	garr_stoermeldungen[st_config.i16_meld_startindex + 10] := FALSE;
	garr_stoermeldungen[st_config.i16_meld_startindex + 11] := FALSE;
	garr_stoermeldungen[st_config.i16_meld_startindex + 12] := FALSE;
	garr_stoermeldungen[st_config.i16_meld_startindex + 13] := FALSE;
	garr_stoermeldungen[st_config.i16_meld_startindex + 14] := FALSE;
	garr_stoermeldungen[st_config.i16_meld_startindex + 15] := FALSE;
	garr_stoermeldungen[st_config.i16_meld_startindex + 16] := FALSE;
	garr_stoermeldungen[st_config.i16_meld_startindex + 17] := FALSE;
	garr_stoermeldungen[st_config.i16_meld_startindex + 18] := FALSE;
	garr_stoermeldungen[st_config.i16_meld_startindex + 19] := FALSE;

	garr_betriebsmeldungen[st_config.i16_meld_startindex + 0] :=FALSE;
	garr_betriebsmeldungen[st_config.i16_meld_startindex + 1] := FALSE;
	garr_betriebsmeldungen[st_config.i16_meld_startindex + 2] := FALSE;
	garr_betriebsmeldungen[st_config.i16_meld_startindex + 3] := FALSE;
	garr_betriebsmeldungen[st_config.i16_meld_startindex + 4] := FALSE;
	garr_betriebsmeldungen[st_config.i16_meld_startindex + 5] := FALSE;
	garr_betriebsmeldungen[st_config.i16_meld_startindex + 6] := FALSE;
	garr_betriebsmeldungen[st_config.i16_meld_startindex + 7] := FALSE;
	garr_betriebsmeldungen[st_config.i16_meld_startindex + 8] := FALSE;
	garr_betriebsmeldungen[st_config.i16_meld_startindex + 9] := FALSE;
	garr_betriebsmeldungen[st_config.i16_meld_startindex + 10] := FALSE;
	garr_betriebsmeldungen[st_config.i16_meld_startindex + 11] := FALSE;
	garr_betriebsmeldungen[st_config.i16_meld_startindex + 12] := FALSE;
	garr_betriebsmeldungen[st_config.i16_meld_startindex + 13] := FALSE;
	garr_betriebsmeldungen[st_config.i16_meld_startindex + 14] := FALSE;
	garr_betriebsmeldungen[st_config.i16_meld_startindex + 15] := FALSE;
	garr_betriebsmeldungen[st_config.i16_meld_startindex + 16] := FALSE;
	garr_betriebsmeldungen[st_config.i16_meld_startindex + 17] := FALSE;
	garr_betriebsmeldungen[st_config.i16_meld_startindex + 18] := FALSE;
	garr_betriebsmeldungen[st_config.i16_meld_startindex + 19] := FALSE;
END_IF
END_PROGRAM
ACTION auto_speichern_laden:
(*========================================================================================*)
(*ohne Timer wurde nicht immer gespeichert*)
fb_ton_end(
	IN:=  i16_auftrag = KEIN_WARTUNG_AUFTRAG,
	PT:= t#100ms,
	Q=> ,
	ET=> );


(*Werkzeug Daten speichern*)
IF	fb_ton_end.Q AND gi16_maschinenstatusinfo <> STATUS_MASCHINE_ARBEITET AND
	(MEMCMP(ADR(st_wartungsprotokoll_wkz_copy.st_wartung_wkz), ADR(gst_datensatz.st_wartungsprotokoll.st_wartung_wkz), SIZEOF(st_wartungsprotokoll_wkz_copy.st_wartung_wkz)) <> 0 ) THEN
	i16_auftrag:=SCHREIBE_WARTUNGSPROTOKOLL_WKZ;
END_IF


(*Maschinen Daten speichern*)
IF	fb_ton_end.Q AND gi16_maschinenstatusinfo <> STATUS_MASCHINE_ARBEITET AND
	(MEMCMP(ADR(st_wartungsprotokoll_md_copy.st_wartung_md), ADR(gst_datensatz.st_wartungsprotokoll.st_wartung_md), SIZEOF(st_wartungsprotokoll_md_copy.st_wartung_md)) <> 0 ) THEN
	i16_auftrag:=SCHREIBE_WARTUNGSPROTOKOLL_MD;
END_IF

(*Button in der Oberfläche für das Reseten nach der Wartung*)
IF fb_ton_end.Q AND gi16_maschinenstatusinfo <> STATUS_MASCHINE_ARBEITET AND fb_r_trig_reset_wkz.Q THEN
	i16_auftrag:=SCHREIBE_WARTUNGSPROTOKOLL_WKZ_RESET;
END_IF
END_ACTION
ACTION fb_Aufrufe:
fb_xml_srv_read(
	sNetId:= ,
	ePath:= PATH_GENERIC,
	nMode:= XMLSRV_SKIPMISSING,
	sFilePath:=sPathName,
	bExecute:= ,
	tTimeout:= t#20s,
	bBusy=> ,
	bError=> ,
	nErrId=> );


fb_xml_srv_write(
	sNetId:= '',
	ePath:= PATH_GENERIC,
	nMode:= XMLSRV_ADDMISSING,
	sFilePath:=sPathName,
	bExecute:= ,
	tTimeout:= t#10s,
	bBusy=> ,
	bError=> ,
	nErrId=> );


fbFindFiles(
	bExecute	:= ,
	sNetId		:= '',
	sPathName	:= sPathName,
	pFindList		:= ADR(file),
	cbFindList	:= SIZEOF(file),
	tTimeout	:= t#1s );


fb_nt_start_process(
	NETID:= '',
	PATHSTR:= 'C:\Windows\System32\wscript.exe',
	DIRNAME:=s_tools_path,
	COMNDLINE:=CONCAT(visu.s_akt_sprache,'_Wartung_nach_server.vbs'),	 	(*CONCAT(visu.s_akt_sprache,'_Wartung_nach_server.vbs'),		'de_Wartung_nach_server.vbs', 	*)
	START:= ,
	TMOUT:= DEFAULT_ADS_TIMEOUT,
	BUSY=> ,
	ERR=> ,
	ERRID=> nErrId);



FB_GetHostName(
	sNetID:= '127.0.0.1.1.1',
	bExecute:= , 
	tTimeout:= , 
	bBusy=> ,
	bError=> ,
	nErrID=> , 
	sHostName=> );
END_ACTION
ACTION FileName_erstellen:
(*Name für Werkzeug Datei*)
sFileName_wkz:='';
sFileName_wkz:=CONCAT(sFileName_wkz,gst_datensatz.st_md.s_aktuelles_wkz);
sFileName_wkz:=CONCAT(sFileName_wkz,s_Trennstelle);
sFileName_wkz:=CONCAT(sFileName_wkz,FB_GetHostName.sHostName);
sFileName_wkz:=CONCAT(sFileName_wkz,s_Trennstelle);
sFileName_wkz:=CONCAT(sFileName_wkz,gstr_datum);

(*Name für Maschinen Datei*)
sFileName_md:='';
sFileName_md:=CONCAT(sFileName_md,FB_GetHostName.sHostName);
sFileName_md:=CONCAT(sFileName_md,'.xml');
END_ACTION
ACTION Zaehler:
IF fb_state_entry.i16_step = BEREIT THEN
	(*Übergabe der aktuellen Betriebsstunden der Zelle in die Wartungsstruktur*)
	gst_datensatz.st_wartungsprotokoll.st_wartung_md.betriebsstunden := gst_datensatz.st_md.i32_betriebssekundenzaehler/ 3600;

	(*Übergabe des aktuellen Hubzählers der Zelle in die Wartungsstruktur*)
	gst_datensatz.st_wartungsprotokoll.st_wartung_md.hubzaehler := gst_datensatz.st_md.i32_bestueckhubzaehler;

	(*Übergabe der aktuell produzierten Stecker der Zelle in die Wartungsstruktur*)
	gst_datensatz.st_wartungsprotokoll.st_wartung_md.produzierte_stecker := gst_datensatz.st_md.produzierte_Stecker;

	(*Übergabe des aktuellen Hubzählers des benutzten Werkzeugs an die Wartungsstruktur*)
	gst_datensatz.st_wartungsprotokoll.st_wartung_wkz.hubzaehler := i32_bestueckhubzaehler_wkz_copy + (gst_datensatz.st_md.i32_bestueckhubzaehler-i32_bestueckhubzaehler_md_copy);
END_IF
END_ACTION

(* POU Gemeinsamkeiten17xx/WT Transport/ST_Hublift_links, ST *)
PROGRAM ST_Hublift_links
VAR_INPUT
	st_config							: struct_config;
	st_ctrl_in							: struct_ctrl_in;
	e_station_nachher_in_erlaubnis		: BOOL := FALSE;
	e_station_nachher_in_angekommen	: BOOL := FALSE;
END_VAR
VAR_IN_OUT
	st_visu							: struct_visu;
END_VAR
VAR_OUTPUT
	st_ctrl_out						: struct_ctrl_out;
	a_station_nachher_out_anforderung	: BOOL := FALSE;
	a_station_nachher_out_abgegeben	: BOOL := FALSE;
END_VAR
VAR
	fb_ton_wz						: TON;
	fb_ton_uez						: TON;
	tb_ton_wt_anwesend				: TON;
	fb_ton_quitt						: TON;
	fb_r_trig_start						: R_TRIG;
	fb_state_entry						: ST_StateEntry;
	sm_kein_wt_anwesend				: BOOL := FALSE;
	sm_keine_busverbindung			: BOOL := FALSE;
	sm_schiebetuere_nicht_geschlossen	: BOOL := FALSE;

	e_sensor_wt_anwesend			AT %I* : BOOL;
	e_sensor_wt_von_fb_eingezogen	AT %I* : BOOL;
	e_wc_state						AT%I*: BOOL;	(* 0=Data valid, 1=Data invalid *)

	e_schiebetuere_geschlossen			AT %I* : BOOL;
	a_lampe_erlaubnis_schiebetuere_oeffnen		AT %Q* : BOOL;	(* Wenn Lampe TRUE dann darf der Bediener die Schiebetüre öffnen *)
END_VAR
(* Zeiten *)
fb_ton_wz(IN:= , PT:= , Q=>  , ET=> );
fb_ton_uez(IN:= , PT:= , Q=>  , ET=> );
tb_ton_wt_anwesend(IN:=e_sensor_wt_anwesend , PT:= t#500ms, Q=>  , ET=> );
fb_ton_quitt(IN:= , PT:= t#100ms, Q=> , ET=> );

(* Flanken *)
fb_r_trig_start(CLK:=ST_Euchner_Handbedienpult.b_Taste_Power , Q=>);

(* Toplevel *)
IF fb_state_entry.i16_next_step > INIT AND fb_state_entry.i16_next_step < FEHLER THEN
	IF fb_state_entry.i16_next_step < STOP THEN
		IF st_ctrl_in.b_stop THEN
			fb_state_entry.i16_next_step := STOP;
		END_IF
	END_IF

	(* Allgemeine Fehler *)
	IF 	st_config.b_station_aktiv AND NOT st_config.b_station_in_simulation AND
		(zyl_hublift_links_lift.st_ctrl.out.b_fehler OR
		zyl_hublift_links_wt_einzug.st_ctrl.out.b_fehler OR
		zyl_hublift_links_wt_klinke.st_ctrl.out.b_fehler OR
		zyl_hublift_links_stopper.st_ctrl.out.b_fehler OR
		zyl_hublift_links_eingriffschutz.st_ctrl.out.b_fehler) THEN
			fb_state_entry.i16_next_step := FEHLER;

	(* Zylinder im Handbetrieb *)
	ELSIF gi16_betriebsart = HAND AND st_config.b_station_aktiv AND NOT st_config.b_station_in_simulation AND
		((st_visu.st_zyl.i16_nr_zyl_im_handbetrieb = zyl_hublift_links_lift.fb.st_config.i16_identnummer) OR
		(st_visu.st_zyl.i16_nr_zyl_im_handbetrieb = zyl_hublift_links_wt_einzug.fb.st_config.i16_identnummer) OR
		(st_visu.st_zyl.i16_nr_zyl_im_handbetrieb = zyl_hublift_links_wt_klinke.fb.st_config.i16_identnummer) OR
		(st_visu.st_zyl.i16_nr_zyl_im_handbetrieb = zyl_hublift_links_stopper.fb.st_config.i16_identnummer)  OR
		(st_visu.st_zyl.i16_nr_zyl_im_handbetrieb = zyl_hublift_links_eingriffschutz.fb.st_config.i16_identnummer) ) THEN
			fb_state_entry.i16_next_step := FEHLER;
	END_IF
END_IF

(* ==================================Schrittkette================================ *)
fb_state_entry(
	i16_next_step:= ,
	i16_pos:= 1,
	s_debugtext:= ,
	E=> ,
	X=> ,
	i16_step=> ,
	i16_last_step=> );

CASE fb_state_entry.i16_step OF
(*=======================================================*)
	INIT_OBJ:
		IF st_config.b_config_fertig THEN
			fb_state_entry.i16_next_step := INIT;
		END_IF

(*=======================================================*)
	INIT:
		IF fb_state_entry.E THEN
			fb_ton_wz.IN := FALSE;
			fb_ton_uez.IN	:= FALSE;
			fb_ton_quitt.IN := FALSE;
			sm_kein_wt_anwesend	:= FALSE;
			sm_keine_busverbindung := FALSE;
			sm_schiebetuere_nicht_geschlossen := FALSE;
			a_station_nachher_out_anforderung := FALSE;
			a_station_nachher_out_abgegeben := FALSE;
			a_lampe_erlaubnis_schiebetuere_oeffnen := FALSE;
			st_ctrl_out.b_fehler := FALSE;
			st_ctrl_out.b_bereit := FALSE;
			st_ctrl_out.b_fertig := FALSE;
			st_ctrl_out.b_kontroller_start := FALSE;
			zyl_hublift_links_lift.st_ctrl.in.b_einfahren := FALSE;
			zyl_hublift_links_lift.st_ctrl.in.b_ausfahren := FALSE;
			zyl_hublift_links_wt_einzug.st_ctrl.in.b_einfahren := FALSE;
			zyl_hublift_links_wt_einzug.st_ctrl.in.b_ausfahren := FALSE;
			zyl_hublift_links_wt_klinke.st_ctrl.in.b_einfahren := FALSE;
			zyl_hublift_links_wt_klinke.st_ctrl.in.b_ausfahren := FALSE;
			zyl_hublift_links_stopper.st_ctrl.in.b_einfahren := FALSE;
			zyl_hublift_links_stopper.st_ctrl.in.b_ausfahren := FALSE;
			zyl_hublift_links_eingriffschutz.st_ctrl.in.b_einfahren := FALSE;
			zyl_hublift_links_eingriffschutz.st_ctrl.in.b_ausfahren := FALSE;
		END_IF

		(*-----------------------Weiterschaltbedingungen----------------------------*)
		IF st_ctrl_in.b_init THEN
			zyl_hublift_links_lift.st_ctrl.in.b_quittieren := FALSE;
			zyl_hublift_links_wt_einzug.st_ctrl.in.b_quittieren := FALSE;
			zyl_hublift_links_wt_klinke.st_ctrl.in.b_quittieren := FALSE;
			zyl_hublift_links_stopper.st_ctrl.in.b_quittieren := FALSE;
			zyl_hublift_links_eingriffschutz.st_ctrl.in.b_quittieren := FALSE;

			IF st_config.b_station_aktiv AND NOT st_config.b_station_in_simulation AND gst_datensatz.st_md.b_wt_transport_aktiv THEN
				fb_state_entry.i16_next_step := 15;
			ELSE
				fb_state_entry.i16_next_step := BEREIT;
			END_IF
		END_IF

(*=======================================================*)
	15: (* Prüfe, ob Busverbindung vorhanden ist *)

		(*-----------------------Weiterschaltbedingungen----------------------------*)
		IF e_wc_state THEN
			sm_keine_busverbindung := TRUE;
			fb_state_entry.i16_next_step := FEHLER;
		ELSE
			fb_state_entry.i16_next_step := 18;
		END_IF

(*=======================================================*)
	18: (* Prüfe, ob Eingriffschutz geschlossen ist *)

		(*-----------------------Weiterschaltbedingungen----------------------------*)
		IF NOT e_schiebetuere_geschlossen THEN
			sm_schiebetuere_nicht_geschlossen := TRUE;
			fb_state_entry.i16_next_step := FEHLER;
		ELSE
			fb_state_entry.i16_next_step := 20;
		END_IF

(*=======================================================*)
	20: (* Initialisierung: Stopper ausfahren *)
		IF fb_state_entry.E THEN
			zyl_hublift_links_stopper.st_ctrl.in.b_ausfahren := TRUE;
		END_IF

		(*-----------------------Weiterschaltbedingungen----------------------------*)
		IF zyl_hublift_links_stopper.st_ctrl.out.b_ausgefahren THEN
			zyl_hublift_links_stopper.st_ctrl.in.b_ausfahren := FALSE;
			fb_state_entry.i16_next_step := 30;
		END_IF

(*=======================================================*)
	30: (* Initialisierung: Abfrage auf WT *)
		IF tb_ton_wt_anwesend.Q THEN
		(* WT anwesend *)
			IF zyl_hublift_links_lift.fb.e_sensor1_eingefahren THEN
			(* Hublift unten *)
				fb_state_entry.i16_next_step := 120;
			ELSE
			(* Hublift oben *)
				fb_state_entry.i16_next_step := 155;
			END_IF
		ELSE
		(* Kein WT vorhanden oder vielleicht steht einer am Stopper *)
			fb_state_entry.i16_next_step := 40;
		END_IF

(*=======================================================*)
	40: (* Initialisierung: Klinke einfahren *)
		IF fb_state_entry.E THEN
			zyl_hublift_links_wt_klinke.st_ctrl.in.b_einfahren := TRUE;
		END_IF

		(*-----------------------Weiterschaltbedingungen----------------------------*)
		IF zyl_hublift_links_wt_klinke.st_ctrl.out.b_eingefahren THEN
			zyl_hublift_links_wt_klinke.st_ctrl.in.b_einfahren := FALSE;
			IF zyl_hublift_links_lift.fb.e_sensor1_eingefahren THEN
			(* Hublift unten *)
				fb_state_entry.i16_next_step := 70;
			ELSE
			(* Hublift oben *)
				fb_state_entry.i16_next_step := 50;
			END_IF
		END_IF

(*=======================================================*)
	50: (* Initialisierung: WT-Einzug einfahren *)
		IF fb_state_entry.E THEN
			zyl_hublift_links_wt_einzug.st_ctrl.in.b_einfahren := TRUE;
		END_IF

		(*-----------------------Weiterschaltbedingungen----------------------------*)
		IF zyl_hublift_links_wt_einzug.st_ctrl.out.b_eingefahren THEN
			zyl_hublift_links_wt_einzug.st_ctrl.in.b_einfahren := FALSE;
			fb_state_entry.i16_next_step := 60;
		END_IF

(*=======================================================*)
	60: (* Initialisierung: Lift einfahren *)
		IF fb_state_entry.E THEN
			zyl_hublift_links_lift.st_ctrl.in.b_einfahren := TRUE;
		END_IF

		(*-----------------------Weiterschaltbedingungen----------------------------*)
		IF zyl_hublift_links_lift.st_ctrl.out.b_eingefahren THEN
			zyl_hublift_links_lift.st_ctrl.in.b_einfahren := FALSE;
			fb_state_entry.i16_next_step := 70;
		END_IF

(*=======================================================*)
	70: (* WT-Einzug ausfahren *)
		IF fb_state_entry.E THEN
			zyl_hublift_links_wt_einzug.st_ctrl.in.b_ausfahren := TRUE;
		END_IF

		(*-----------------------Weiterschaltbedingungen----------------------------*)
		IF zyl_hublift_links_wt_einzug.st_ctrl.out.b_ausgefahren THEN
			zyl_hublift_links_wt_einzug.st_ctrl.in.b_ausfahren := FALSE;
			fb_state_entry.i16_next_step := 80;
		END_IF

(*=======================================================*)
	80: (* Initialisierung: Stopper einfahren *)
		IF fb_state_entry.E THEN
			zyl_hublift_links_stopper.st_ctrl.in.b_einfahren := TRUE;
		END_IF

		(*-----------------------Weiterschaltbedingungen----------------------------*)
		IF zyl_hublift_links_stopper.st_ctrl.out.b_eingefahren THEN
			zyl_hublift_links_stopper.st_ctrl.in.b_einfahren := FALSE;
			fb_state_entry.i16_next_step := 90;
		END_IF

(*=======================================================*)
	90: (* Eingriffschutz ausfahren*)
		IF fb_state_entry.E THEN
			zyl_hublift_links_eingriffschutz.st_ctrl.in.b_ausfahren := TRUE;
		END_IF

		(*-----------------------Weiterschaltbedingungen----------------------------*)
		IF zyl_hublift_links_eingriffschutz.st_ctrl.out.b_ausgefahren THEN
			zyl_hublift_links_eingriffschutz.st_ctrl.in.b_ausfahren := FALSE;
			fb_state_entry.i16_next_step := BEREIT;
		END_IF

(*=======================================================*)
	BEREIT:
		IF fb_state_entry.E THEN
			st_ctrl_out.b_bereit := TRUE;
		END_IF

		(*-----------------------Weiterschaltbedingungen----------------------------*)
		IF st_config.b_station_aktiv AND NOT st_config.b_station_in_simulation AND gst_datensatz.st_md.b_wt_transport_aktiv THEN
			(* Hublift und WT Transport aktiv *)
			fb_state_entry.i16_next_step := 110;
		ELSIF NOT st_config.b_station_aktiv AND st_config.b_station_in_simulation AND gst_datensatz.st_md.b_wt_transport_aktiv THEN
			(* Simulation des Hubliftes *)
			fb_state_entry.i16_next_step := 160;
		ELSE
			;(* Hublift und WT Transport NICHT aktiv *)
		END_IF

(*=======================================================*)
	110:	(* Warte bis der WT angekommen ist *)

		(*-----------------------Weiterschaltbedingungen----------------------------*)
		IF tb_ton_wt_anwesend.Q THEN
			fb_state_entry.i16_next_step := 120;
		END_IF

(*=======================================================*)
	120: (* Klinke ausfahren -> WT einhaken*)
		IF fb_state_entry.E THEN
			zyl_hublift_links_wt_klinke.st_ctrl.in.b_ausfahren := TRUE;
		END_IF

		(*-----------------------Weiterschaltbedingungen----------------------------*)
		IF zyl_hublift_links_wt_klinke.st_ctrl.out.b_ausgefahren AND
			e_sensor_wt_anwesend THEN
			zyl_hublift_links_wt_klinke.st_ctrl.in.b_ausfahren := FALSE;
			fb_state_entry.i16_next_step := 130;
		END_IF

(*=======================================================*)
	130: (* WT-Einzug einfahren und Stopper bei Signal ausfahren *)
		IF fb_state_entry.E THEN
			zyl_hublift_links_wt_einzug.st_ctrl.in.b_einfahren := TRUE;
		END_IF

		(*-----------------------Weiterschaltbedingungen----------------------------*)
		IF 	e_sensor_wt_von_fb_eingezogen OR
			zyl_hublift_links_wt_einzug.st_ctrl.out.b_eingefahren THEN
				zyl_hublift_links_stopper.st_ctrl.in.b_ausfahren := TRUE;
				fb_state_entry.i16_next_step := 140;
		END_IF

(*=======================================================*)
	140: (* WT-Einzug ist eingefahren und Stopper ist ausgefahren *)

		(*-----------------------Weiterschaltbedingungen----------------------------*)
		IF 	zyl_hublift_links_stopper.st_ctrl.out.b_ausgefahren AND
			zyl_hublift_links_wt_einzug.st_ctrl.out.b_eingefahren AND
			e_sensor_wt_anwesend THEN
				zyl_hublift_links_stopper.st_ctrl.in.b_ausfahren := FALSE;
				zyl_hublift_links_wt_einzug.st_ctrl.in.b_einfahren := FALSE;
				fb_state_entry.i16_next_step := 150;
		END_IF

(*=======================================================*)
	150: (* WT mit Lift anheben *)
		IF fb_state_entry.E THEN
			zyl_hublift_links_lift.st_ctrl.in.b_ausfahren := TRUE;
		END_IF

		(*-----------------------Weiterschaltbedingungen----------------------------*)
		IF zyl_hublift_links_lift.st_ctrl.out.b_ausgefahren THEN
			zyl_hublift_links_lift.st_ctrl.in.b_ausfahren := FALSE;
			fb_state_entry.i16_next_step := 155;
		END_IF

(*=======================================================*)
	155: (* Warte auf Simulation oder Taste_Power *)
		IF fb_state_entry.E THEN
			a_lampe_erlaubnis_schiebetuere_oeffnen := TRUE;
		END_IF

		(*-----------------------Weiterschaltbedingungen----------------------------*)
		IF st_config.b_station_in_simulation OR
			(fb_r_trig_start.Q AND e_schiebetuere_geschlossen) THEN
			fb_state_entry.i16_next_step := 160;
		END_IF

		IF fb_state_entry.X THEN
			a_lampe_erlaubnis_schiebetuere_oeffnen := FALSE;
		END_IF

(*=======================================================*)
	160: (* Warte auf Folgestation *)
		IF fb_state_entry.E THEN
			st_ctrl_out.b_bereit := TRUE;
			a_station_nachher_out_anforderung := TRUE;
		END_IF

		(*-----------------------Weiterschaltbedingungen----------------------------*)
		IF  e_station_nachher_in_erlaubnis AND NOT fb_state_entry.E THEN
			a_station_nachher_out_anforderung := FALSE;
			IF st_config.b_station_in_simulation THEN
				fb_state_entry.i16_next_step := 180;
			ELSE
				IF e_sensor_wt_anwesend THEN
					fb_state_entry.i16_next_step := 165;
				ELSE
					fb_state_entry.i16_next_step := 190;
				END_IF
			END_IF
		END_IF

(*=======================================================*)
	165: (* Eingriffschutz einfahren*)
		IF fb_state_entry.E THEN
			zyl_hublift_links_eingriffschutz.st_ctrl.in.b_einfahren := TRUE;
		END_IF

		(*-----------------------Weiterschaltbedingungen----------------------------*)
		IF zyl_hublift_links_eingriffschutz.st_ctrl.out.b_eingefahren THEN
			zyl_hublift_links_eingriffschutz.st_ctrl.in.b_einfahren := FALSE;
			fb_state_entry.i16_next_step := 170;
		END_IF

(*=======================================================*)
	170: (* WT-Einzug ausfahren und Klinke einfahren und WT aushaken *)
		IF fb_state_entry.E THEN
			zyl_hublift_links_wt_einzug.st_ctrl.in.b_ausfahren := TRUE;
			zyl_hublift_links_wt_klinke.st_ctrl.in.b_einfahren := TRUE;
			st_ctrl_out.b_kontroller_start := TRUE;
		END_IF

		(*-----------------------Weiterschaltbedingungen----------------------------*)
		IF 	zyl_hublift_links_wt_einzug.st_ctrl.out.b_ausgefahren AND
			zyl_hublift_links_wt_klinke.st_ctrl.out.b_eingefahren
			THEN
				st_ctrl_out.b_kontroller_start := FALSE;
				zyl_hublift_links_wt_einzug.st_ctrl.in.b_ausfahren := FALSE;
				zyl_hublift_links_wt_klinke.st_ctrl.in.b_einfahren := FALSE;
				fb_state_entry.i16_next_step := 180;
		END_IF

(*=======================================================*)
	180:	(* Warte bis WT angekommen ist *)
		IF fb_state_entry.E THEN
			a_station_nachher_out_abgegeben := TRUE;
		END_IF

		(*-----------------------Weiterschaltbedingungen----------------------------*)
		IF e_station_nachher_in_angekommen THEN
			a_station_nachher_out_abgegeben := FALSE;
			IF st_config.b_station_in_simulation THEN
				fb_state_entry.i16_next_step := BEREIT;
			ELSE
				fb_state_entry.i16_next_step := 185;
			END_IF
		END_IF

(*=======================================================*)
	185: (* Eingriffschutz ausfahren*)
		IF fb_state_entry.E THEN
			zyl_hublift_links_eingriffschutz.st_ctrl.in.b_ausfahren := TRUE;
		END_IF

		(*-----------------------Weiterschaltbedingungen----------------------------*)
		IF zyl_hublift_links_eingriffschutz.st_ctrl.out.b_ausgefahren THEN
			zyl_hublift_links_eingriffschutz.st_ctrl.in.b_ausfahren := FALSE;
			fb_state_entry.i16_next_step := 190;
		END_IF

(*=======================================================*)
	190: (* Klinke einfahren*)
		IF fb_state_entry.E THEN
			zyl_hublift_links_wt_klinke.st_ctrl.in.b_einfahren := TRUE;
		END_IF

		(*-----------------------Weiterschaltbedingungen----------------------------*)
		IF zyl_hublift_links_wt_klinke.st_ctrl.out.b_eingefahren THEN
			zyl_hublift_links_wt_klinke.st_ctrl.in.b_einfahren := FALSE;
			fb_state_entry.i16_next_step := 200;
		END_IF

(*=======================================================*)
	200: (* WT-Einzug einfahren  *)
		IF fb_state_entry.E THEN
			zyl_hublift_links_wt_einzug.st_ctrl.in.b_einfahren := TRUE;
		END_IF

		(*-----------------------Weiterschaltbedingungen----------------------------*)
		IF zyl_hublift_links_wt_einzug.st_ctrl.out.b_eingefahren THEN
			zyl_hublift_links_wt_einzug.st_ctrl.in.b_einfahren := FALSE;
			fb_state_entry.i16_next_step := 210;
		END_IF

(*=======================================================*)
	210: (*  Lift einfahren *)
		IF fb_state_entry.E THEN
			zyl_hublift_links_lift.st_ctrl.in.b_einfahren := TRUE;
		END_IF

		(*-----------------------Weiterschaltbedingungen----------------------------*)
		IF zyl_hublift_links_lift.st_ctrl.out.b_eingefahren THEN
			zyl_hublift_links_lift.st_ctrl.in.b_einfahren := FALSE;
			fb_state_entry.i16_next_step := 220;
		END_IF

(*=======================================================*)
	220: (* WT-Einzug ausfahren  *)
		IF fb_state_entry.E THEN
			zyl_hublift_links_wt_einzug.st_ctrl.in.b_ausfahren := TRUE;
		END_IF

		(*-----------------------Weiterschaltbedingungen----------------------------*)
		IF zyl_hublift_links_wt_einzug.st_ctrl.out.b_ausgefahren THEN
			zyl_hublift_links_wt_einzug.st_ctrl.in.b_ausfahren := FALSE;
			fb_state_entry.i16_next_step := 230;
		END_IF

(*=======================================================*)
	230: (* Stopper einfahren *)
		IF fb_state_entry.E THEN
			zyl_hublift_links_stopper.st_ctrl.in.b_einfahren := TRUE;
		END_IF

		(*-----------------------Weiterschaltbedingungen----------------------------*)
		IF zyl_hublift_links_stopper.st_ctrl.out.b_eingefahren THEN
			zyl_hublift_links_stopper.st_ctrl.in.b_einfahren := FALSE;
			fb_state_entry.i16_next_step := BEREIT;
		END_IF

(*=======================================================*)
	FEHLER:
		IF fb_state_entry.E THEN
			st_ctrl_out.b_fehler := TRUE;
			fb_ton_quitt.IN := FALSE;
			a_station_nachher_out_anforderung := FALSE;
			a_station_nachher_out_abgegeben := FALSE;
			zyl_hublift_links_lift.st_ctrl.in.b_quittieren := FALSE;
			zyl_hublift_links_wt_einzug.st_ctrl.in.b_quittieren := FALSE;
			zyl_hublift_links_wt_klinke.st_ctrl.in.b_quittieren := FALSE;
			zyl_hublift_links_stopper.st_ctrl.in.b_quittieren := FALSE;
			zyl_hublift_links_eingriffschutz.st_ctrl.in.b_quittieren := FALSE;
		END_IF

		(*-----------------------Weiterschaltbedingungen----------------------------*)
		IF st_ctrl_in.b_quitt AND NOT fb_state_entry.E THEN
			st_ctrl_out.b_fehler := FALSE;
			zyl_hublift_links_lift.st_ctrl.in.b_quittieren := TRUE;
			zyl_hublift_links_wt_einzug.st_ctrl.in.b_quittieren := TRUE;
			zyl_hublift_links_wt_klinke.st_ctrl.in.b_quittieren := TRUE;
			zyl_hublift_links_stopper.st_ctrl.in.b_quittieren := TRUE;
			zyl_hublift_links_eingriffschutz.st_ctrl.in.b_quittieren := TRUE;
			fb_ton_quitt.IN := TRUE;
		END_IF

		IF fb_ton_quitt.Q THEN
			fb_ton_quitt.IN := FALSE;
			fb_state_entry.i16_next_step := INIT;
		END_IF

(*=======================================================*)
	STOP:
		IF fb_state_entry.E THEN
			fb_ton_quitt.IN := FALSE;
			zyl_hublift_links_lift.st_ctrl.in.b_quittieren := FALSE;
			zyl_hublift_links_wt_einzug.st_ctrl.in.b_quittieren := FALSE;
			zyl_hublift_links_wt_klinke.st_ctrl.in.b_quittieren := FALSE;
			zyl_hublift_links_stopper.st_ctrl.in.b_quittieren := FALSE;
			zyl_hublift_links_eingriffschutz.st_ctrl.in.b_quittieren := FALSE;
		END_IF

		(*-----------------------Weiterschaltbedingungen----------------------------*)
		IF st_ctrl_in.b_quitt AND NOT fb_state_entry.E THEN
			fb_ton_quitt.IN := TRUE;
			zyl_hublift_links_lift.st_ctrl.in.b_quittieren := TRUE;
			zyl_hublift_links_wt_einzug.st_ctrl.in.b_quittieren := TRUE;
			zyl_hublift_links_wt_klinke.st_ctrl.in.b_quittieren := TRUE;
			zyl_hublift_links_stopper.st_ctrl.in.b_quittieren := TRUE;
			zyl_hublift_links_eingriffschutz.st_ctrl.in.b_quittieren := TRUE;
		END_IF

		IF fb_ton_quitt.Q THEN
			fb_ton_quitt.IN := FALSE;
			fb_state_entry.i16_next_step := INIT;
		END_IF
END_CASE

fb_state_entry(
	i16_next_step:= ,
	i16_pos:= 2,
	s_debugtext:= ,
	E=> ,
	X=> , 
	i16_step=> ,
	i16_last_step=> );

IF st_config.b_config_fertig THEN
	(* Fehlermeldungen und Betriebsmeldungen ab dem Startindex in die globalen Meldungsarrays schreiben *)
	garr_stoermeldungen[st_config.i16_meld_startindex + 0] := sm_kein_wt_anwesend;
	garr_stoermeldungen[st_config.i16_meld_startindex + 1] := sm_keine_busverbindung;
	garr_stoermeldungen[st_config.i16_meld_startindex + 2] := sm_schiebetuere_nicht_geschlossen;
	garr_stoermeldungen[st_config.i16_meld_startindex + 3] := FALSE;
	garr_stoermeldungen[st_config.i16_meld_startindex + 4] := FALSE;
	garr_stoermeldungen[st_config.i16_meld_startindex + 5] := FALSE;
	garr_stoermeldungen[st_config.i16_meld_startindex + 6] := FALSE;
	garr_stoermeldungen[st_config.i16_meld_startindex + 7] := FALSE;
	garr_stoermeldungen[st_config.i16_meld_startindex + 8] := FALSE;
	garr_stoermeldungen[st_config.i16_meld_startindex + 9] := FALSE;
	garr_stoermeldungen[st_config.i16_meld_startindex + 10] := FALSE;
	garr_stoermeldungen[st_config.i16_meld_startindex + 11] := FALSE;
	garr_stoermeldungen[st_config.i16_meld_startindex + 12] := FALSE;
	garr_stoermeldungen[st_config.i16_meld_startindex + 13] := FALSE;
	garr_stoermeldungen[st_config.i16_meld_startindex + 14] := FALSE;
	garr_stoermeldungen[st_config.i16_meld_startindex + 15] := FALSE;
	garr_stoermeldungen[st_config.i16_meld_startindex + 16] := FALSE;
	garr_stoermeldungen[st_config.i16_meld_startindex + 17] := FALSE;
	garr_stoermeldungen[st_config.i16_meld_startindex + 18] := FALSE;
	garr_stoermeldungen[st_config.i16_meld_startindex + 19] := FALSE;
	
